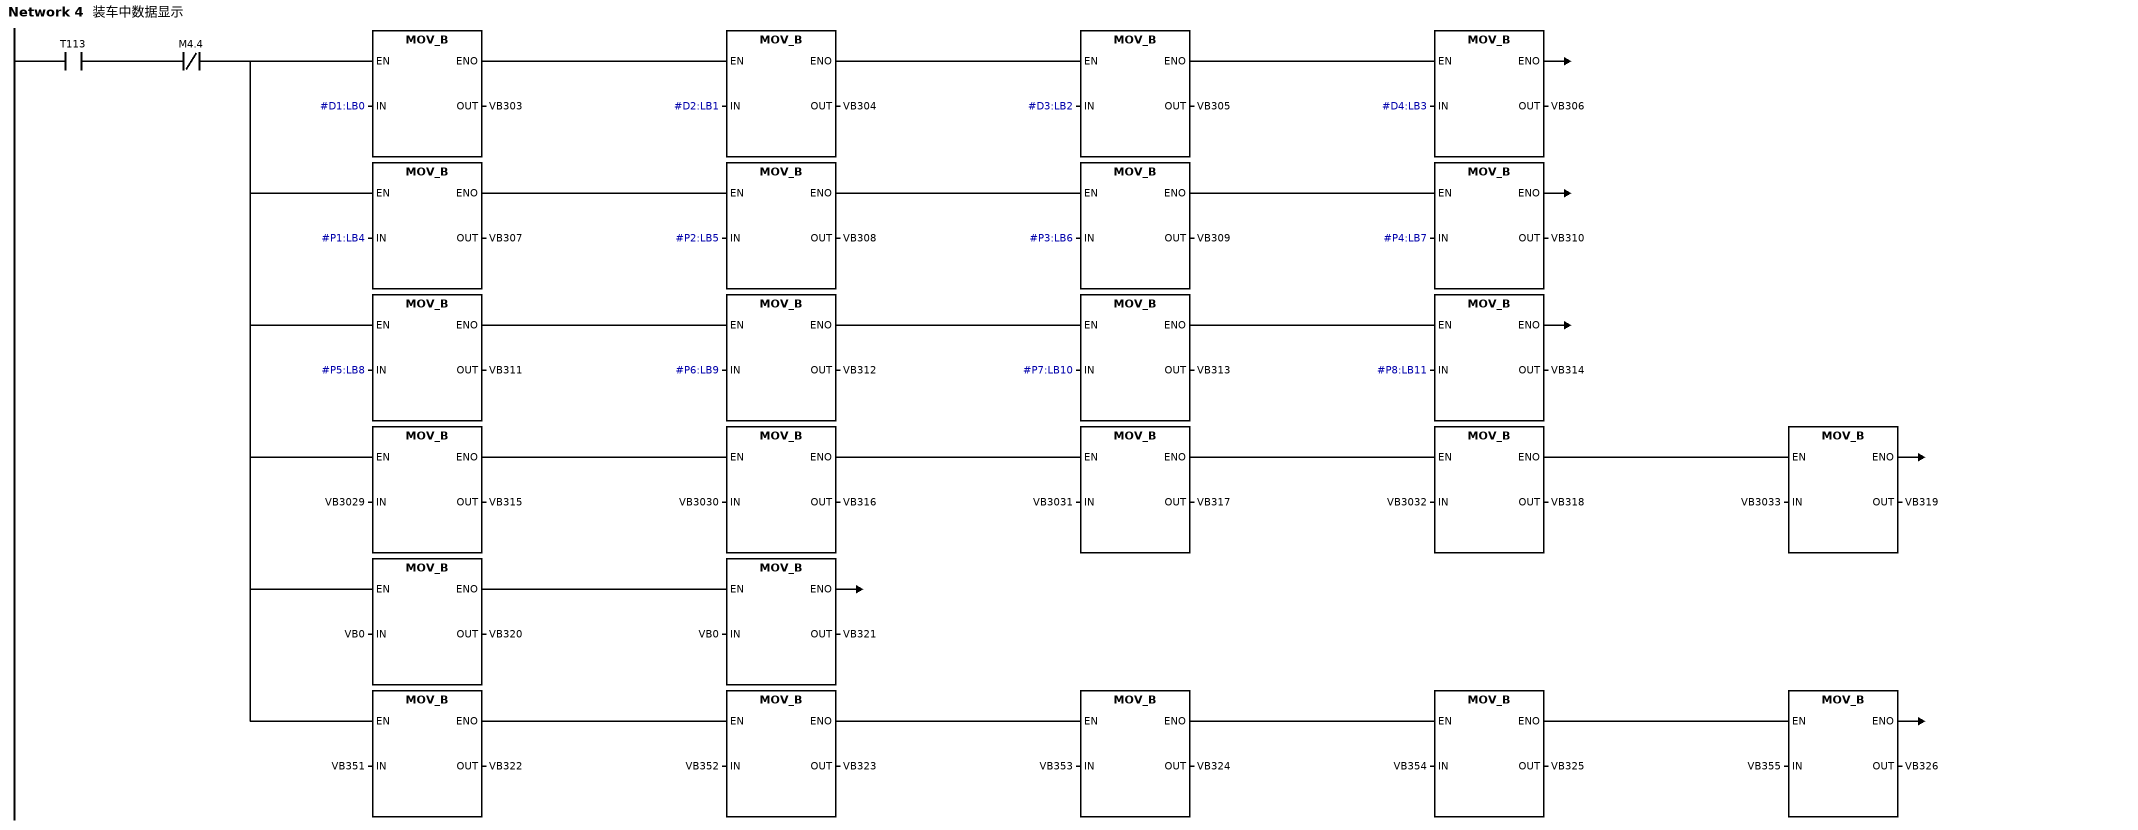
[picture p24: SBR13 networks 4-4]
Network 4 // 装车中数据显示
LD     T113
AN     M4.4
LPS
MOVB   #D1:LB0, VB303
AENO
MOVB   #D2:LB1, VB304
AENO
MOVB   #D3:LB2, VB305
AENO
MOVB   #D4:LB3, VB306
LRD
MOVB   #P1:LB4, VB307
AENO
MOVB   #P2:LB5, VB308
AENO
MOVB   #P3:LB6, VB309
AENO
MOVB   #P4:LB7, VB310
LRD
MOVB   #P5:LB8, VB311
AENO
MOVB   #P6:LB9, VB312
AENO
MOVB   #P7:LB10, VB313
AENO
MOVB   #P8:LB11, VB314
LRD
MOVB   VB3029, VB315
AENO
MOVB   VB3030, VB316
AENO
MOVB   VB3031, VB317
AENO
MOVB   VB3032, VB318
AENO
MOVB   VB3033, VB319
LRD
MOVB   VB0, VB320
AENO
MOVB   VB0, VB321
LPP
MOVB   VB351, VB322
AENO
MOVB   VB352, VB323
AENO
MOVB   VB353, VB324
AENO
MOVB   VB354, VB325
AENO
MOVB   VB355, VB326
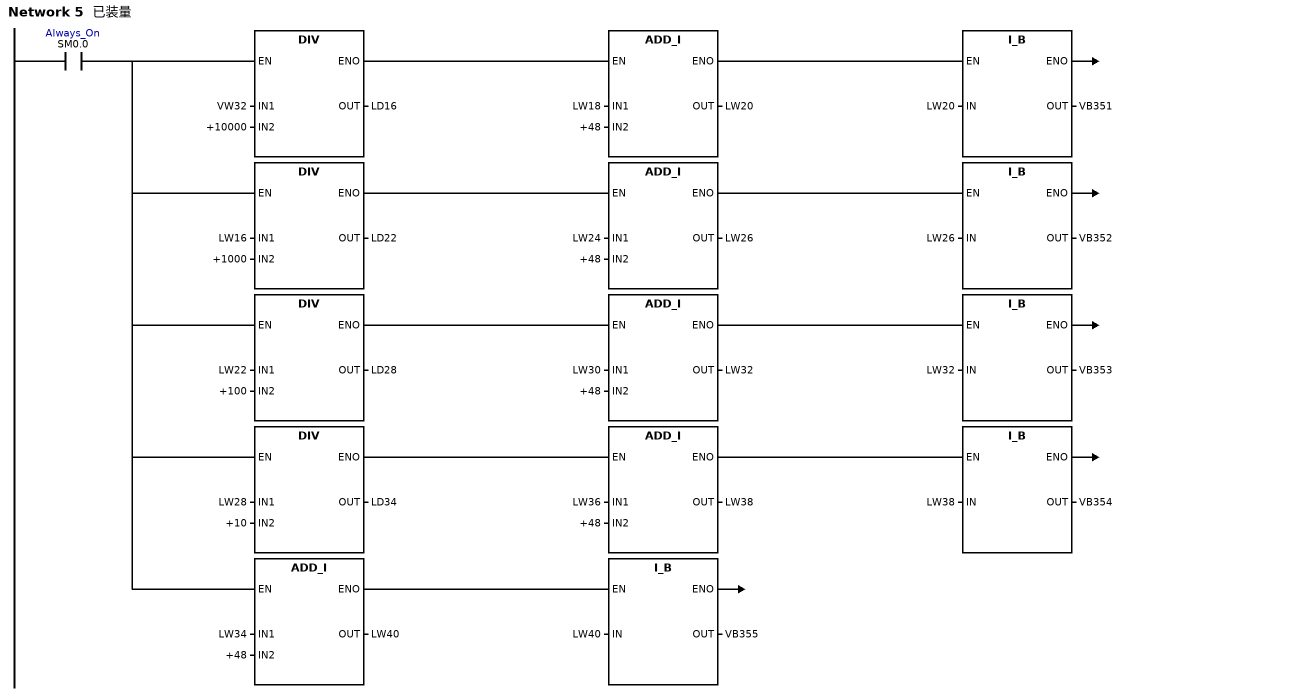
Network 5 // 已装量
LD     Always_On:SM0.0
LPS
MOVW   VW32, LW18
AENO
DIV    +10000, LD16
AENO
MOVW   LW18, LW20
AENO
+I     +48, LW20
AENO
ITB    LW20, VB351
LRD
MOVW   LW16, LW24
AENO
DIV    +1000, LD22
AENO
MOVW   LW24, LW26
AENO
+I     +48, LW26
AENO
ITB    LW26, VB352
LRD
MOVW   LW22, LW30
AENO
DIV    +100, LD28
AENO
MOVW   LW30, LW32
AENO
+I     +48, LW32
AENO
ITB    LW32, VB353
LRD
MOVW   LW28, LW36
AENO
DIV    +10, LD34
AENO
MOVW   LW36, LW38
AENO
+I     +48, LW38
AENO
ITB    LW38, VB354
LPP
MOVW   LW34, LW40
AENO
+I     +48, LW40
AENO
ITB    LW40, VB355
END_SUBROUTINE_BLOCK

SUBROUTINE_BLOCK LED4:SBR14
TITLE=
VAR_INPUT
D1:BYTE;	// LB0 
D2:BYTE;	// LB1 
D3:BYTE;	// LB2 
D4:BYTE;	// LB3 
P1:BYTE;	// LB4 
P2:BYTE;	// LB5 
P3:BYTE;	// LB6 
P4:BYTE;	// LB7 
P5:BYTE;	// LB8 
P6:BYTE;	// LB9 
P7:BYTE;	// LB10 
P8:BYTE;	// LB11 
RUN:WORD;	// LW12 
END_VAR
BEGIN
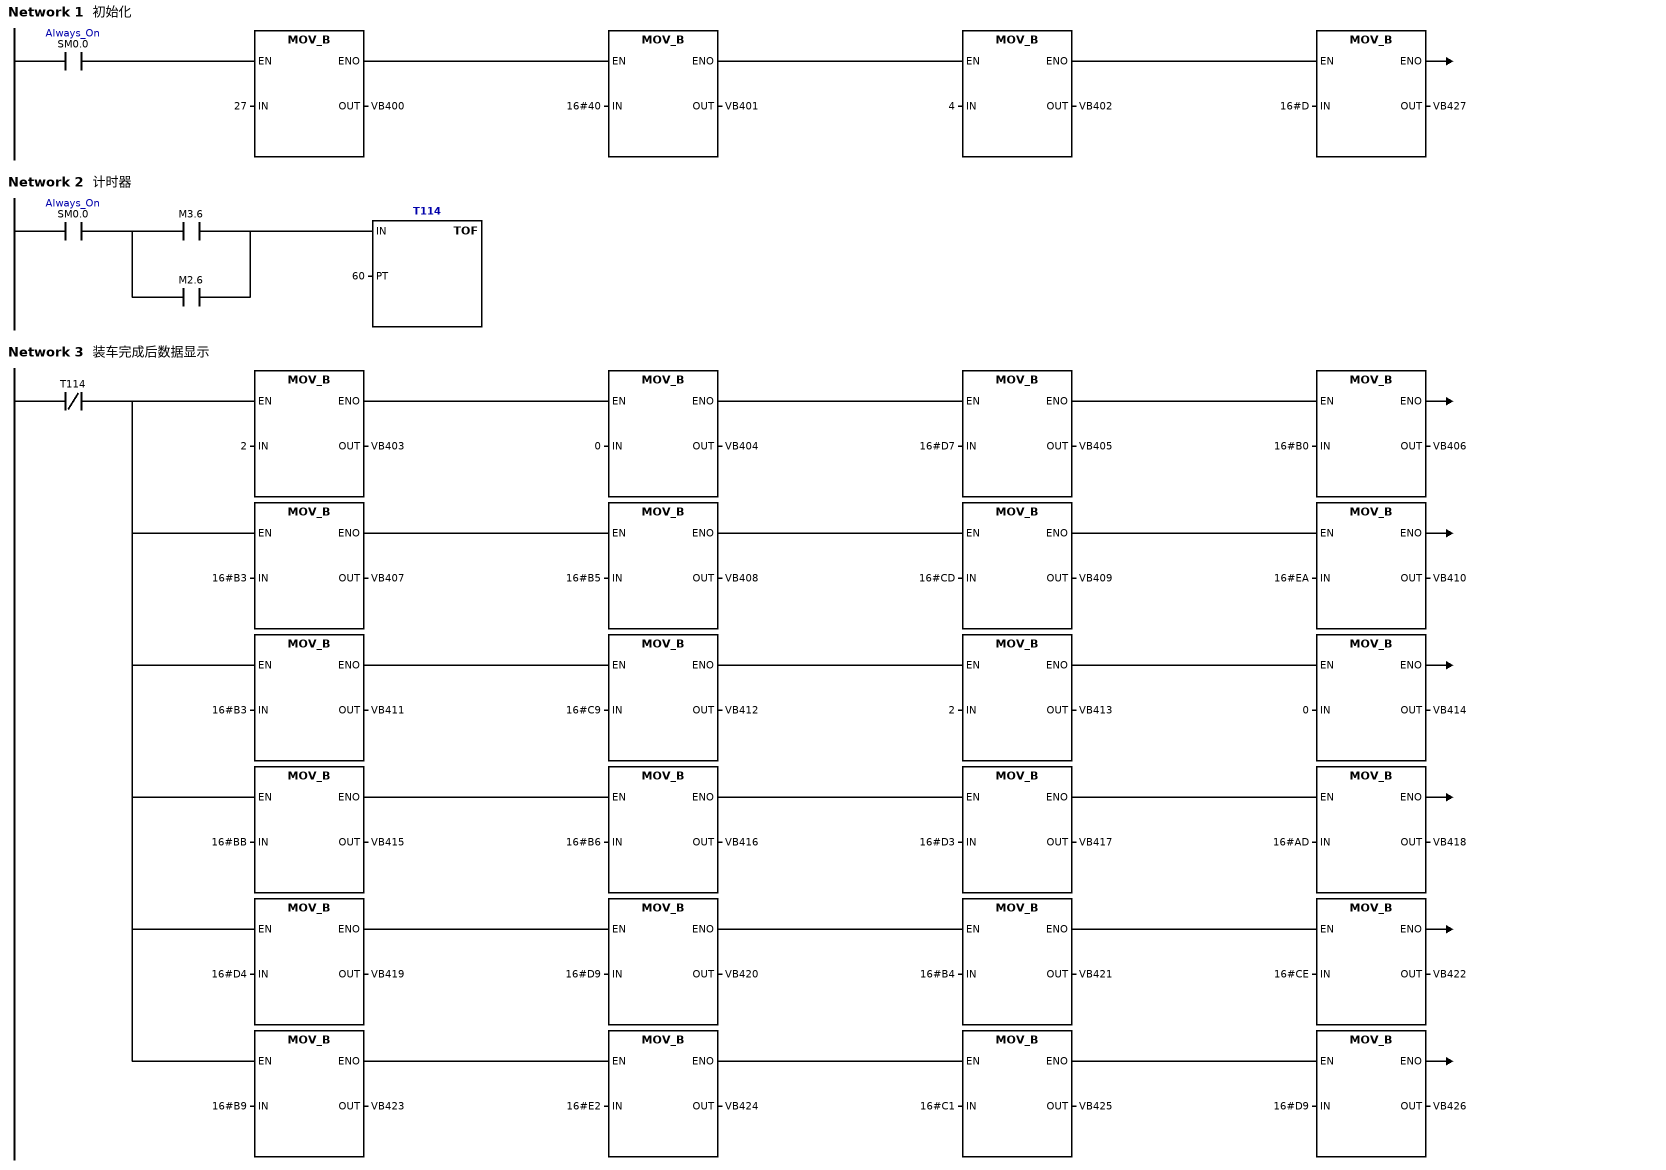
Network 1 // 初始化
LD     Always_On:SM0.0
MOVB   27, VB400
AENO
MOVB   16#40, VB401
AENO
MOVB   4, VB402
AENO
MOVB   16#D, VB427
Network 2 // 计时器
LD     Always_On:SM0.0
LD     M3.6
O      M2.6
ALD
TOF    T114, 60
Network 3 // 装车完成后数据显示
LDN    T114
LPS
MOVB   2, VB403
AENO
MOVB   0, VB404
AENO
MOVB   16#D7, VB405
AENO
MOVB   16#B0, VB406
LRD
MOVB   16#B3, VB407
AENO
MOVB   16#B5, VB408
AENO
MOVB   16#CD, VB409
AENO
MOVB   16#EA, VB410
LRD
MOVB   16#B3, VB411
AENO
MOVB   16#C9, VB412
AENO
MOVB   2, VB413
AENO
MOVB   0, VB414
LRD
MOVB   16#BB, VB415
AENO
MOVB   16#B6, VB416
AENO
MOVB   16#D3, VB417
AENO
MOVB   16#AD, VB418
LRD
MOVB   16#D4, VB419
AENO
MOVB   16#D9, VB420
AENO
MOVB   16#B4, VB421
AENO
MOVB   16#CE, VB422
LPP
MOVB   16#B9, VB423
AENO
MOVB   16#E2, VB424
AENO
MOVB   16#C1, VB425
AENO
MOVB   16#D9, VB426
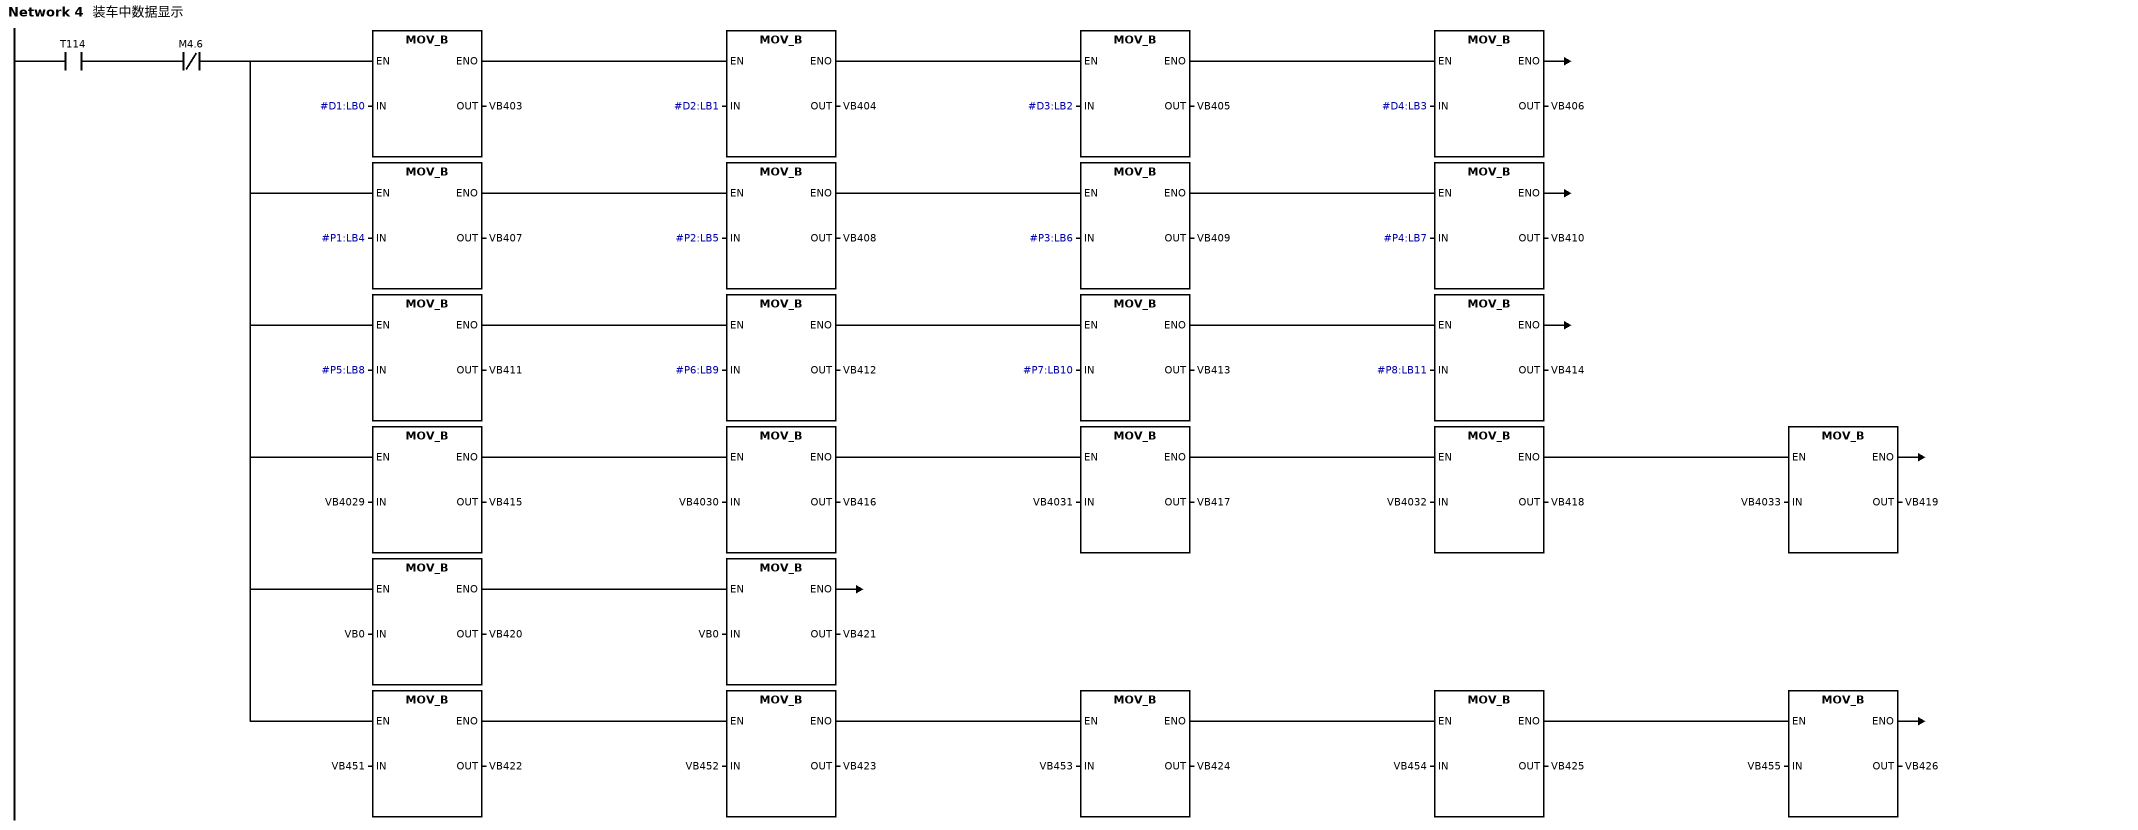
Network 4 // 装车中数据显示
LD     T114
AN     M4.6
LPS
MOVB   #D1:LB0, VB403
AENO
MOVB   #D2:LB1, VB404
AENO
MOVB   #D3:LB2, VB405
AENO
MOVB   #D4:LB3, VB406
LRD
MOVB   #P1:LB4, VB407
AENO
MOVB   #P2:LB5, VB408
AENO
MOVB   #P3:LB6, VB409
AENO
MOVB   #P4:LB7, VB410
LRD
MOVB   #P5:LB8, VB411
AENO
MOVB   #P6:LB9, VB412
AENO
MOVB   #P7:LB10, VB413
AENO
MOVB   #P8:LB11, VB414
LRD
MOVB   VB4029, VB415
AENO
MOVB   VB4030, VB416
AENO
MOVB   VB4031, VB417
AENO
MOVB   VB4032, VB418
AENO
MOVB   VB4033, VB419
LRD
MOVB   VB0, VB420
AENO
MOVB   VB0, VB421
LPP
MOVB   VB451, VB422
AENO
MOVB   VB452, VB423
AENO
MOVB   VB453, VB424
AENO
MOVB   VB454, VB425
AENO
MOVB   VB455, VB426
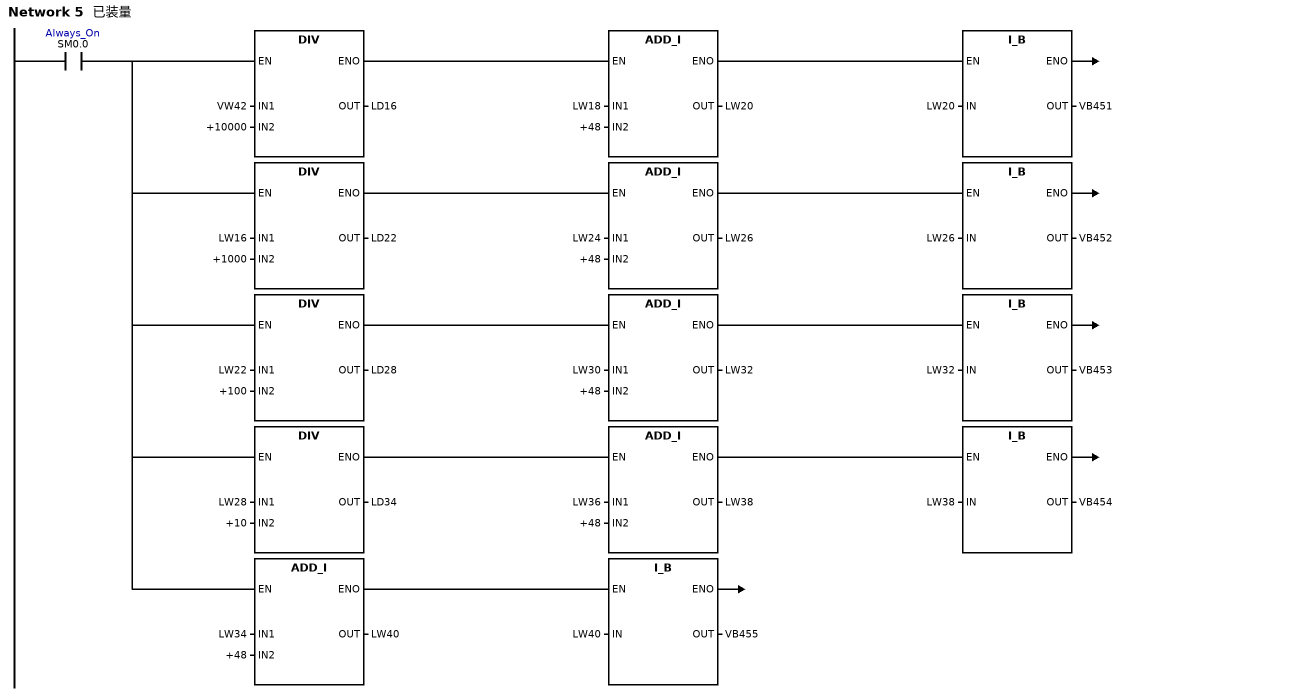
Network 5 // 已装量
LD     Always_On:SM0.0
LPS
MOVW   VW42, LW18
AENO
DIV    +10000, LD16
AENO
MOVW   LW18, LW20
AENO
+I     +48, LW20
AENO
ITB    LW20, VB451
LRD
MOVW   LW16, LW24
AENO
DIV    +1000, LD22
AENO
MOVW   LW24, LW26
AENO
+I     +48, LW26
AENO
ITB    LW26, VB452
LRD
MOVW   LW22, LW30
AENO
DIV    +100, LD28
AENO
MOVW   LW30, LW32
AENO
+I     +48, LW32
AENO
ITB    LW32, VB453
LRD
MOVW   LW28, LW36
AENO
DIV    +10, LD34
AENO
MOVW   LW36, LW38
AENO
+I     +48, LW38
AENO
ITB    LW38, VB454
LPP
MOVW   LW34, LW40
AENO
+I     +48, LW40
AENO
ITB    LW40, VB455
END_SUBROUTINE_BLOCK

SUBROUTINE_BLOCK N1收:SBR21
TITLE=
VAR_OUTPUT
总袋数1:WORD;	// LW0 
袋长1:WORD;	// LW2 
END_VAR
VAR
TEMP1:WORD;	// LW4 
TEMP2:WORD;	// LW6 
TEMP3:WORD;	// LW8 
TEMP4:WORD;	// LW10 
TEMP5:WORD;	// LW12 
TEMP6:WORD;	// LW14 
TEMP7:WORD;	// LW16 
TEMP8:WORD;	// LW18 
TEMP9:WORD;	// LW20 
TEMP10:WORD;	// LW22 
TEMP11:WORD;	// LW24 
TEMP12:WORD;	// LW26 
TEMP13:WORD;	// LW28 
TEMP14:WORD;	// LW30 
TEMP15:WORD;	// LW32 
TEMP16:WORD;	// LW34 
TEMP17:WORD;	// LW36 
TEMP18:WORD;	// LW38 
TEMP19:WORD;	// LW40 
TEMP20:WORD;	// LW42 
TEMP21:WORD;	// LW44 
END_VAR
BEGIN
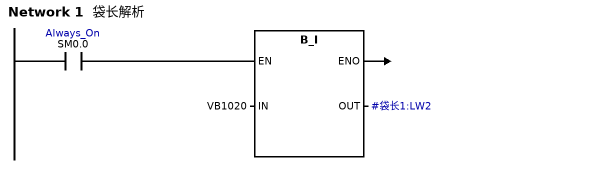
Network 1 // 袋长解析
LD     Always_On:SM0.0
BTI    VB1020, #袋长1:LW2
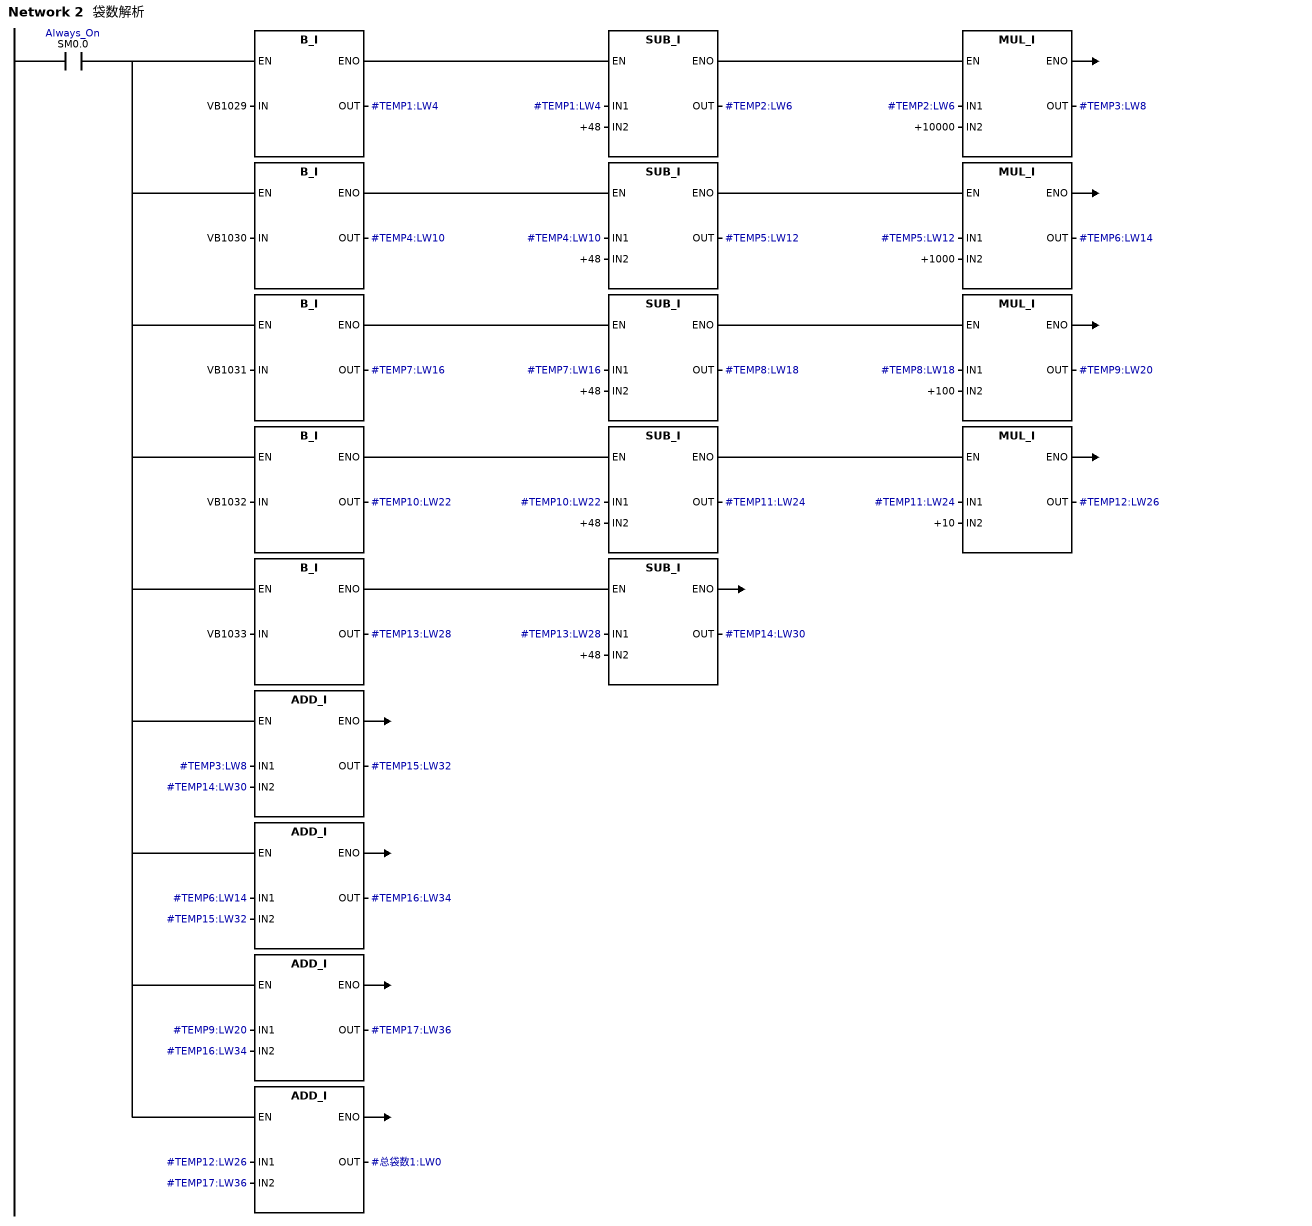
Network 2 // 袋数解析
LD     Always_On:SM0.0
LPS
BTI    VB1029, #TEMP1:LW4
AENO
MOVW   #TEMP1:LW4, #TEMP2:LW6
AENO
-I     +48, #TEMP2:LW6
AENO
MOVW   #TEMP2:LW6, #TEMP3:LW8
*I     +10000, #TEMP3:LW8
LRD
BTI    VB1030, #TEMP4:LW10
AENO
MOVW   #TEMP4:LW10, #TEMP5:LW12
AENO
-I     +48, #TEMP5:LW12
AENO
MOVW   #TEMP5:LW12, #TEMP6:LW14
*I     +1000, #TEMP6:LW14
LRD
BTI    VB1031, #TEMP7:LW16
AENO
MOVW   #TEMP7:LW16, #TEMP8:LW18
AENO
-I     +48, #TEMP8:LW18
AENO
MOVW   #TEMP8:LW18, #TEMP9:LW20
*I     +100, #TEMP9:LW20
LRD
BTI    VB1032, #TEMP10:LW22
AENO
MOVW   #TEMP10:LW22, #TEMP11:LW24
AENO
-I     +48, #TEMP11:LW24
AENO
MOVW   #TEMP11:LW24, #TEMP12:LW26
*I     +10, #TEMP12:LW26
LRD
BTI    VB1033, #TEMP13:LW28
AENO
MOVW   #TEMP13:LW28, #TEMP14:LW30
-I     +48, #TEMP14:LW30
LRD
MOVW   #TEMP3:LW8, #TEMP15:LW32
+I     #TEMP14:LW30, #TEMP15:LW32
LRD
MOVW   #TEMP6:LW14, #TEMP16:LW34
+I     #TEMP15:LW32, #TEMP16:LW34
LRD
MOVW   #TEMP9:LW20, #TEMP17:LW36
+I     #TEMP16:LW34, #TEMP17:LW36
LPP
MOVW   #TEMP12:LW26, #总袋数1:LW0
+I     #TEMP17:LW36, #总袋数1:LW0
END_SUBROUTINE_BLOCK

SUBROUTINE_BLOCK N2收:SBR22
TITLE=
VAR_OUTPUT
总袋数1:WORD;	// LW0 
袋长1:WORD;	// LW2 
END_VAR
VAR
TEMP1:WORD;	// LW4 
TEMP2:WORD;	// LW6 
TEMP3:WORD;	// LW8 
TEMP4:WORD;	// LW10 
TEMP5:WORD;	// LW12 
TEMP6:WORD;	// LW14 
TEMP7:WORD;	// LW16 
TEMP8:WORD;	// LW18 
TEMP9:WORD;	// LW20 
TEMP10:WORD;	// LW22 
TEMP11:WORD;	// LW24 
TEMP12:WORD;	// LW26 
TEMP13:WORD;	// LW28 
TEMP14:WORD;	// LW30 
TEMP15:WORD;	// LW32 
TEMP16:WORD;	// LW34 
TEMP17:WORD;	// LW36 
TEMP18:WORD;	// LW38 
TEMP19:WORD;	// LW40 
TEMP20:WORD;	// LW42 
TEMP21:WORD;	// LW44 
END_VAR
BEGIN
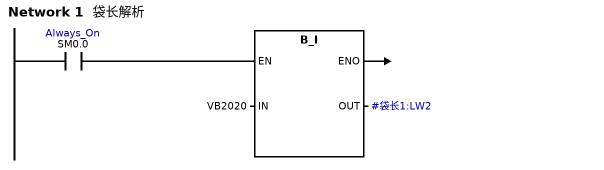
Network 1 // 袋长解析
LD     Always_On:SM0.0
BTI    VB2020, #袋长1:LW2
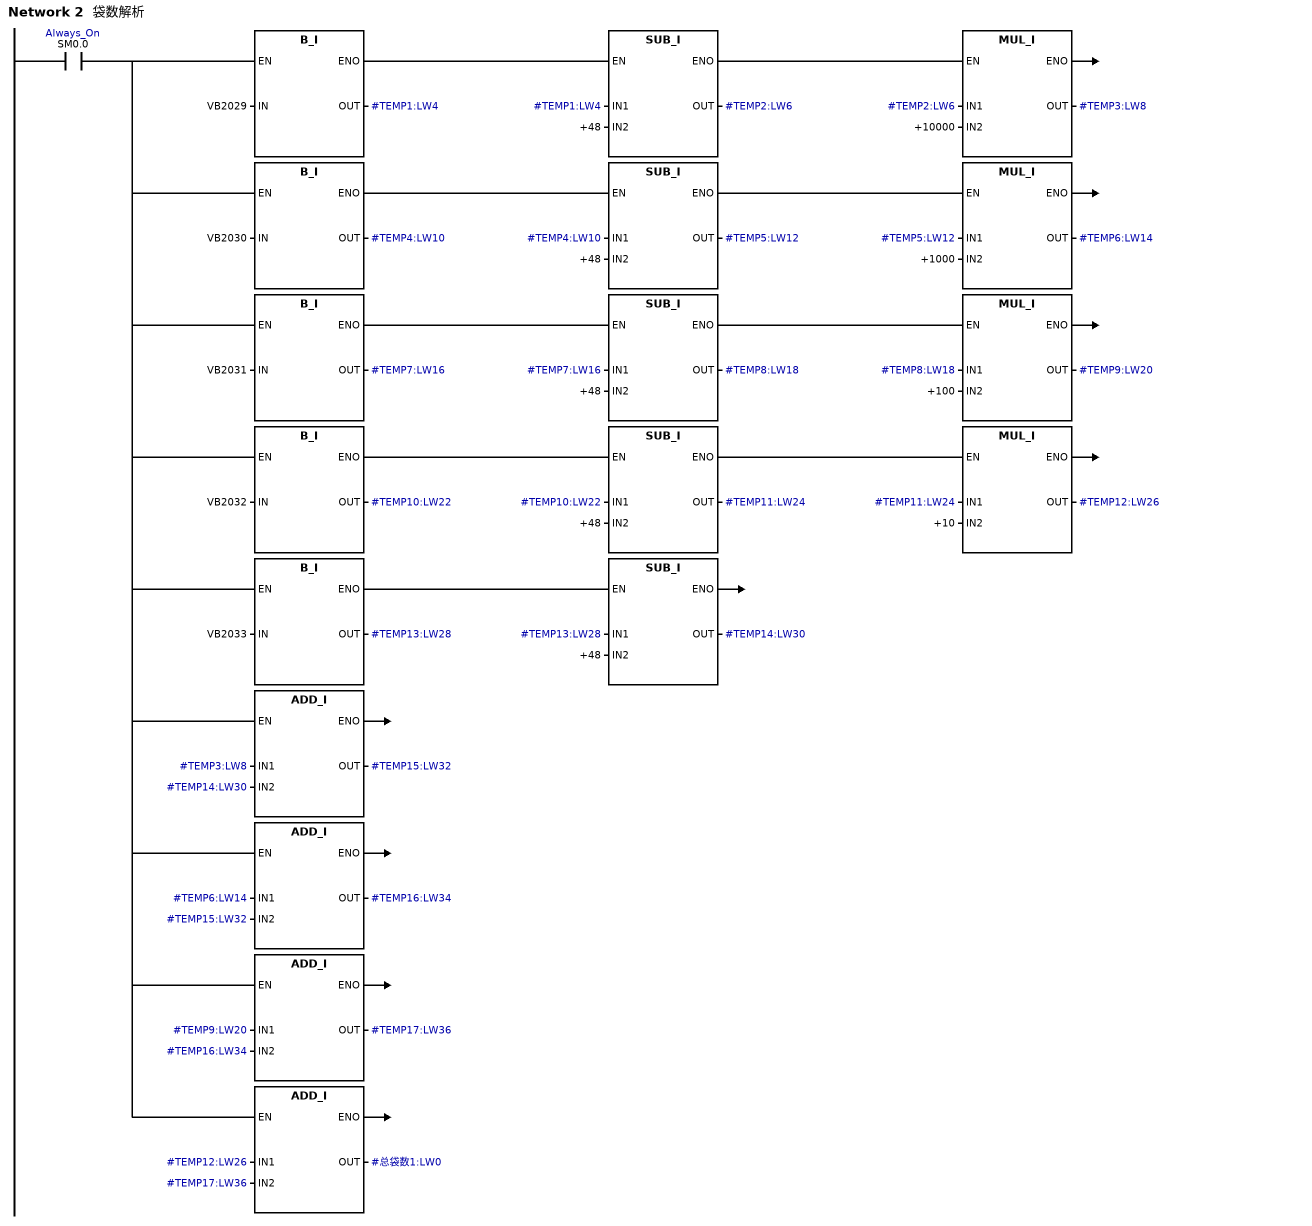
Network 2 // 袋数解析
LD     Always_On:SM0.0
LPS
BTI    VB2029, #TEMP1:LW4
AENO
MOVW   #TEMP1:LW4, #TEMP2:LW6
AENO
-I     +48, #TEMP2:LW6
AENO
MOVW   #TEMP2:LW6, #TEMP3:LW8
*I     +10000, #TEMP3:LW8
LRD
BTI    VB2030, #TEMP4:LW10
AENO
MOVW   #TEMP4:LW10, #TEMP5:LW12
AENO
-I     +48, #TEMP5:LW12
AENO
MOVW   #TEMP5:LW12, #TEMP6:LW14
*I     +1000, #TEMP6:LW14
LRD
BTI    VB2031, #TEMP7:LW16
AENO
MOVW   #TEMP7:LW16, #TEMP8:LW18
AENO
-I     +48, #TEMP8:LW18
AENO
MOVW   #TEMP8:LW18, #TEMP9:LW20
*I     +100, #TEMP9:LW20
LRD
BTI    VB2032, #TEMP10:LW22
AENO
MOVW   #TEMP10:LW22, #TEMP11:LW24
AENO
-I     +48, #TEMP11:LW24
AENO
MOVW   #TEMP11:LW24, #TEMP12:LW26
*I     +10, #TEMP12:LW26
LRD
BTI    VB2033, #TEMP13:LW28
AENO
MOVW   #TEMP13:LW28, #TEMP14:LW30
-I     +48, #TEMP14:LW30
LRD
MOVW   #TEMP3:LW8, #TEMP15:LW32
+I     #TEMP14:LW30, #TEMP15:LW32
LRD
MOVW   #TEMP6:LW14, #TEMP16:LW34
+I     #TEMP15:LW32, #TEMP16:LW34
LRD
MOVW   #TEMP9:LW20, #TEMP17:LW36
+I     #TEMP16:LW34, #TEMP17:LW36
LPP
MOVW   #TEMP12:LW26, #总袋数1:LW0
+I     #TEMP17:LW36, #总袋数1:LW0
END_SUBROUTINE_BLOCK

SUBROUTINE_BLOCK N3收:SBR23
TITLE=
VAR_OUTPUT
总袋数1:WORD;	// LW0 
袋长1:WORD;	// LW2 
END_VAR
VAR
TEMP1:WORD;	// LW4 
TEMP2:WORD;	// LW6 
TEMP3:WORD;	// LW8 
TEMP4:WORD;	// LW10 
TEMP5:WORD;	// LW12 
TEMP6:WORD;	// LW14 
TEMP7:WORD;	// LW16 
TEMP8:WORD;	// LW18 
TEMP9:WORD;	// LW20 
TEMP10:WORD;	// LW22 
TEMP11:WORD;	// LW24 
TEMP12:WORD;	// LW26 
TEMP13:WORD;	// LW28 
TEMP14:WORD;	// LW30 
TEMP15:WORD;	// LW32 
TEMP16:WORD;	// LW34 
TEMP17:WORD;	// LW36 
TEMP18:WORD;	// LW38 
TEMP19:WORD;	// LW40 
TEMP20:WORD;	// LW42 
TEMP21:WORD;	// LW44 
END_VAR
BEGIN
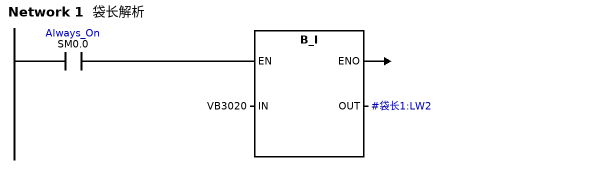
Network 1 // 袋长解析
LD     Always_On:SM0.0
BTI    VB3020, #袋长1:LW2
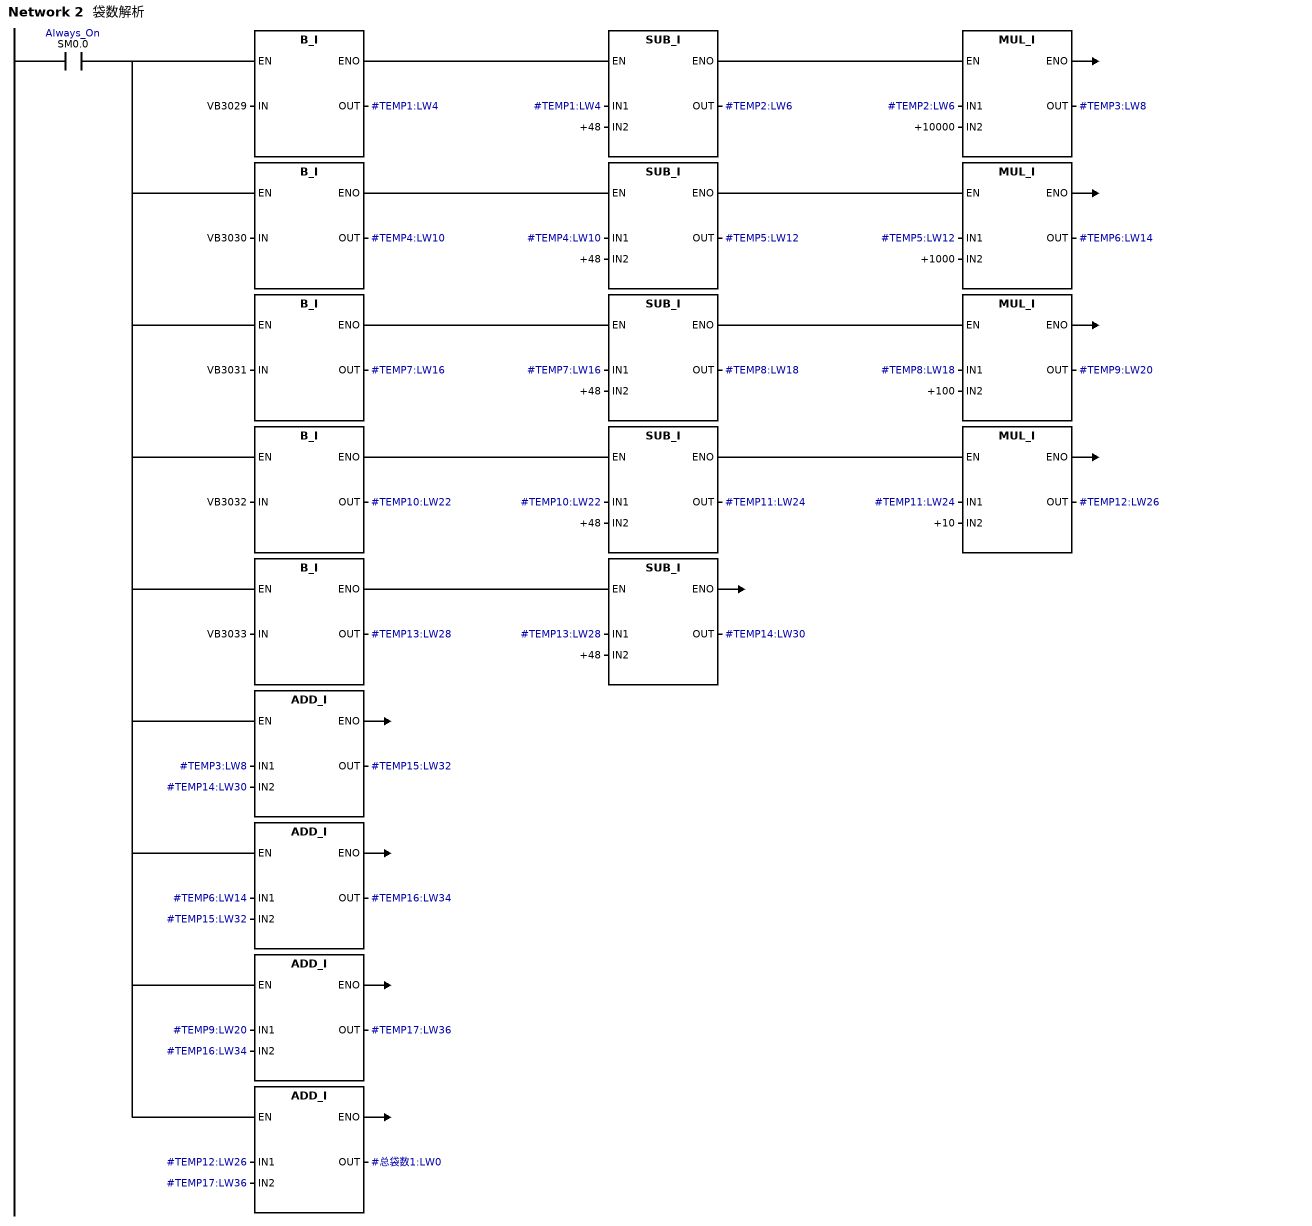
Network 2 // 袋数解析
LD     Always_On:SM0.0
LPS
BTI    VB3029, #TEMP1:LW4
AENO
MOVW   #TEMP1:LW4, #TEMP2:LW6
AENO
-I     +48, #TEMP2:LW6
AENO
MOVW   #TEMP2:LW6, #TEMP3:LW8
*I     +10000, #TEMP3:LW8
LRD
BTI    VB3030, #TEMP4:LW10
AENO
MOVW   #TEMP4:LW10, #TEMP5:LW12
AENO
-I     +48, #TEMP5:LW12
AENO
MOVW   #TEMP5:LW12, #TEMP6:LW14
*I     +1000, #TEMP6:LW14
LRD
BTI    VB3031, #TEMP7:LW16
AENO
MOVW   #TEMP7:LW16, #TEMP8:LW18
AENO
-I     +48, #TEMP8:LW18
AENO
MOVW   #TEMP8:LW18, #TEMP9:LW20
*I     +100, #TEMP9:LW20
LRD
BTI    VB3032, #TEMP10:LW22
AENO
MOVW   #TEMP10:LW22, #TEMP11:LW24
AENO
-I     +48, #TEMP11:LW24
AENO
MOVW   #TEMP11:LW24, #TEMP12:LW26
*I     +10, #TEMP12:LW26
LRD
BTI    VB3033, #TEMP13:LW28
AENO
MOVW   #TEMP13:LW28, #TEMP14:LW30
-I     +48, #TEMP14:LW30
LRD
MOVW   #TEMP3:LW8, #TEMP15:LW32
+I     #TEMP14:LW30, #TEMP15:LW32
LRD
MOVW   #TEMP6:LW14, #TEMP16:LW34
+I     #TEMP15:LW32, #TEMP16:LW34
LRD
MOVW   #TEMP9:LW20, #TEMP17:LW36
+I     #TEMP16:LW34, #TEMP17:LW36
LPP
MOVW   #TEMP12:LW26, #总袋数1:LW0
+I     #TEMP17:LW36, #总袋数1:LW0
END_SUBROUTINE_BLOCK

SUBROUTINE_BLOCK N4收:SBR24
TITLE=
VAR_OUTPUT
总袋数1:WORD;	// LW0 
袋长1:WORD;	// LW2 
END_VAR
VAR
TEMP1:WORD;	// LW4 
TEMP2:WORD;	// LW6 
TEMP3:WORD;	// LW8 
TEMP4:WORD;	// LW10 
TEMP5:WORD;	// LW12 
TEMP6:WORD;	// LW14 
TEMP7:WORD;	// LW16 
TEMP8:WORD;	// LW18 
TEMP9:WORD;	// LW20 
TEMP10:WORD;	// LW22 
TEMP11:WORD;	// LW24 
TEMP12:WORD;	// LW26 
TEMP13:WORD;	// LW28 
TEMP14:WORD;	// LW30 
TEMP15:WORD;	// LW32 
TEMP16:WORD;	// LW34 
TEMP17:WORD;	// LW36 
TEMP18:WORD;	// LW38 
TEMP19:WORD;	// LW40 
TEMP20:WORD;	// LW42 
TEMP21:WORD;	// LW44 
END_VAR
BEGIN
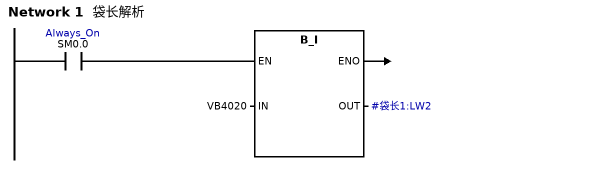
Network 1 // 袋长解析
LD     Always_On:SM0.0
BTI    VB4020, #袋长1:LW2
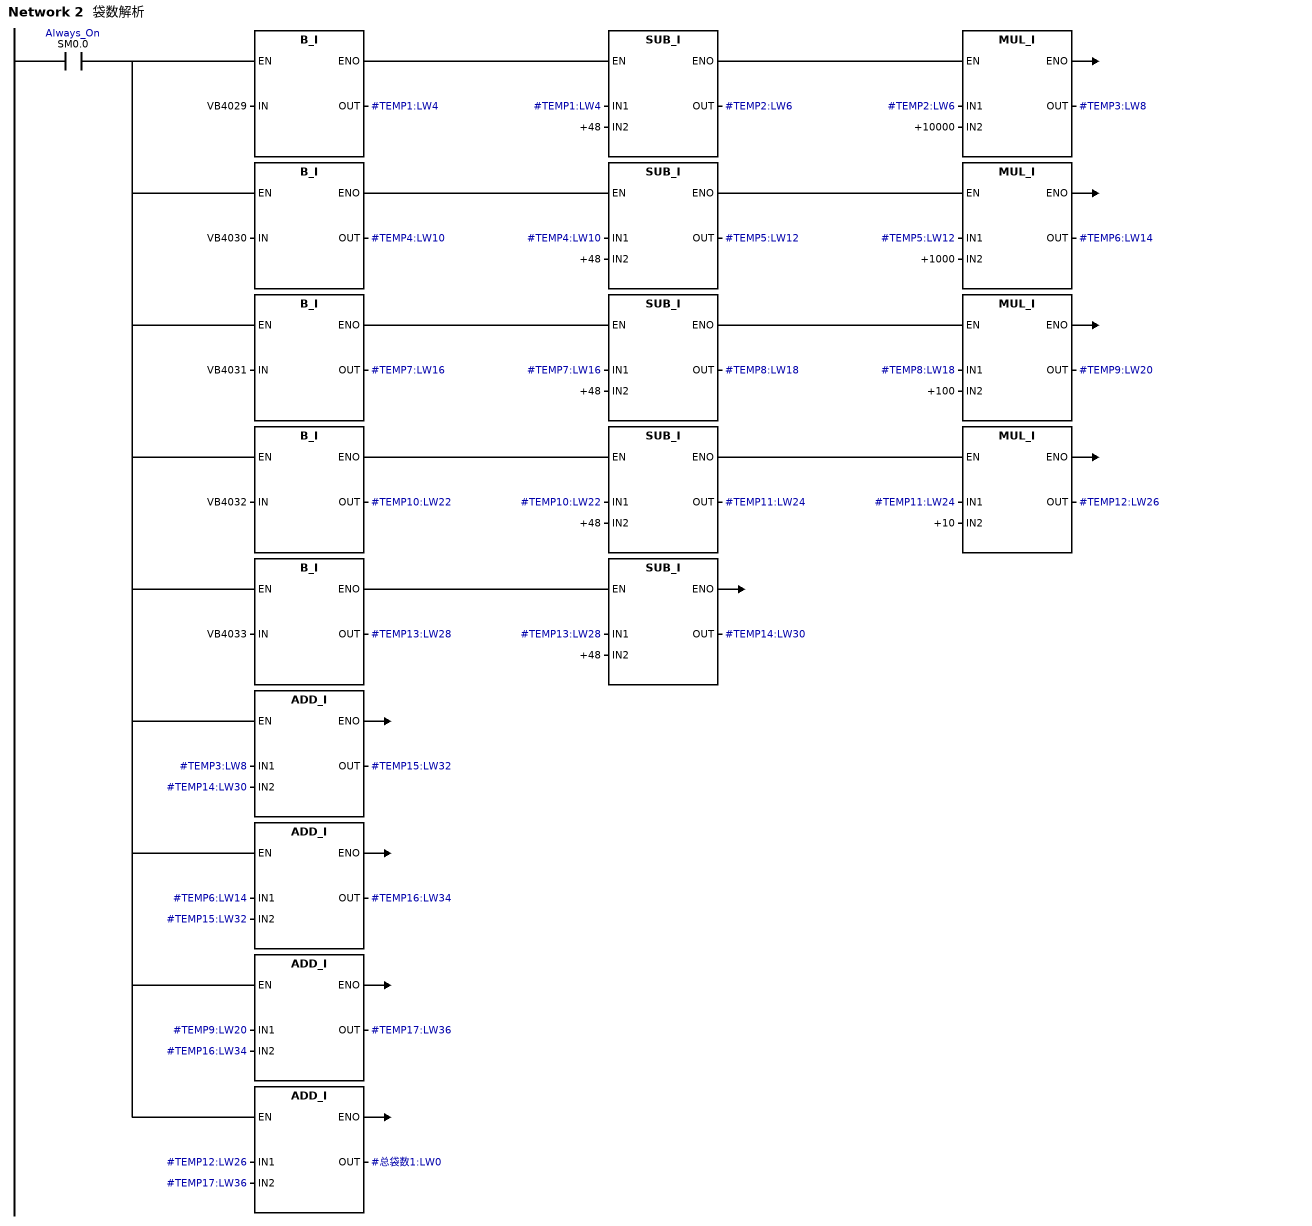
Network 2 // 袋数解析
LD     Always_On:SM0.0
LPS
BTI    VB4029, #TEMP1:LW4
AENO
MOVW   #TEMP1:LW4, #TEMP2:LW6
AENO
-I     +48, #TEMP2:LW6
AENO
MOVW   #TEMP2:LW6, #TEMP3:LW8
*I     +10000, #TEMP3:LW8
LRD
BTI    VB4030, #TEMP4:LW10
AENO
MOVW   #TEMP4:LW10, #TEMP5:LW12
AENO
-I     +48, #TEMP5:LW12
AENO
MOVW   #TEMP5:LW12, #TEMP6:LW14
*I     +1000, #TEMP6:LW14
LRD
BTI    VB4031, #TEMP7:LW16
AENO
MOVW   #TEMP7:LW16, #TEMP8:LW18
AENO
-I     +48, #TEMP8:LW18
AENO
MOVW   #TEMP8:LW18, #TEMP9:LW20
*I     +100, #TEMP9:LW20
LRD
BTI    VB4032, #TEMP10:LW22
AENO
MOVW   #TEMP10:LW22, #TEMP11:LW24
AENO
-I     +48, #TEMP11:LW24
AENO
MOVW   #TEMP11:LW24, #TEMP12:LW26
*I     +10, #TEMP12:LW26
LRD
BTI    VB4033, #TEMP13:LW28
AENO
MOVW   #TEMP13:LW28, #TEMP14:LW30
-I     +48, #TEMP14:LW30
LRD
MOVW   #TEMP3:LW8, #TEMP15:LW32
+I     #TEMP14:LW30, #TEMP15:LW32
LRD
MOVW   #TEMP6:LW14, #TEMP16:LW34
+I     #TEMP15:LW32, #TEMP16:LW34
LRD
MOVW   #TEMP9:LW20, #TEMP17:LW36
+I     #TEMP16:LW34, #TEMP17:LW36
LPP
MOVW   #TEMP12:LW26, #总袋数1:LW0
+I     #TEMP17:LW36, #总袋数1:LW0
END_SUBROUTINE_BLOCK

SUBROUTINE_BLOCK GGLED1_2:SBR31
TITLE=子程序注释
VAR_INPUT
屏3地址:BYTE;	// LB0 
END_VAR
BEGIN
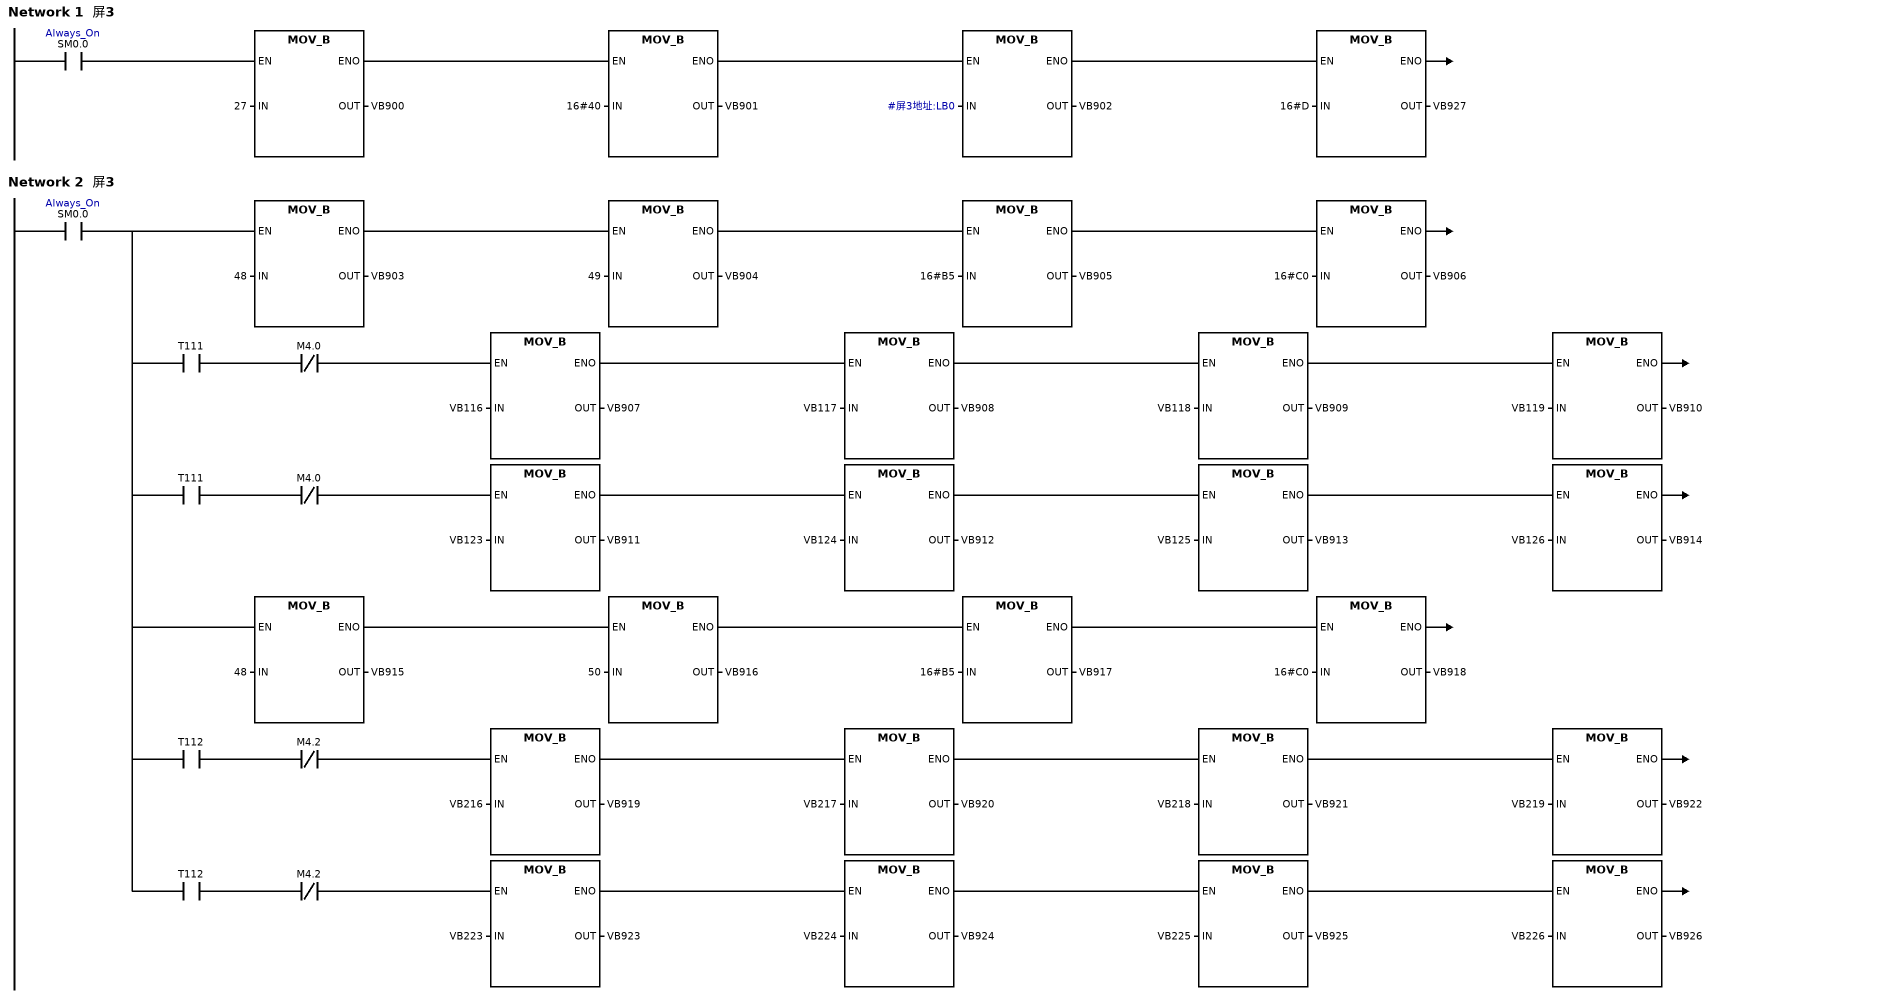
Network 1 // 屏3
LD     Always_On:SM0.0
MOVB   27, VB900
AENO
MOVB   16#40, VB901
AENO
MOVB   #屏3地址:LB0, VB902
AENO
MOVB   16#D, VB927
Network 2 // 屏3
LD     Always_On:SM0.0
LPS
MOVB   48, VB903
AENO
MOVB   49, VB904
AENO
MOVB   16#B5, VB905
AENO
MOVB   16#C0, VB906
LRD
A      T111
AN     M4.0
MOVB   VB116, VB907
AENO
MOVB   VB117, VB908
AENO
MOVB   VB118, VB909
AENO
MOVB   VB119, VB910
LRD
A      T111
AN     M4.0
MOVB   VB123, VB911
AENO
MOVB   VB124, VB912
AENO
MOVB   VB125, VB913
AENO
MOVB   VB126, VB914
LRD
MOVB   48, VB915
AENO
MOVB   50, VB916
AENO
MOVB   16#B5, VB917
AENO
MOVB   16#C0, VB918
LRD
A      T112
AN     M4.2
MOVB   VB216, VB919
AENO
MOVB   VB217, VB920
AENO
MOVB   VB218, VB921
AENO
MOVB   VB219, VB922
LPP
A      T112
AN     M4.2
MOVB   VB223, VB923
AENO
MOVB   VB224, VB924
AENO
MOVB   VB225, VB925
AENO
MOVB   VB226, VB926
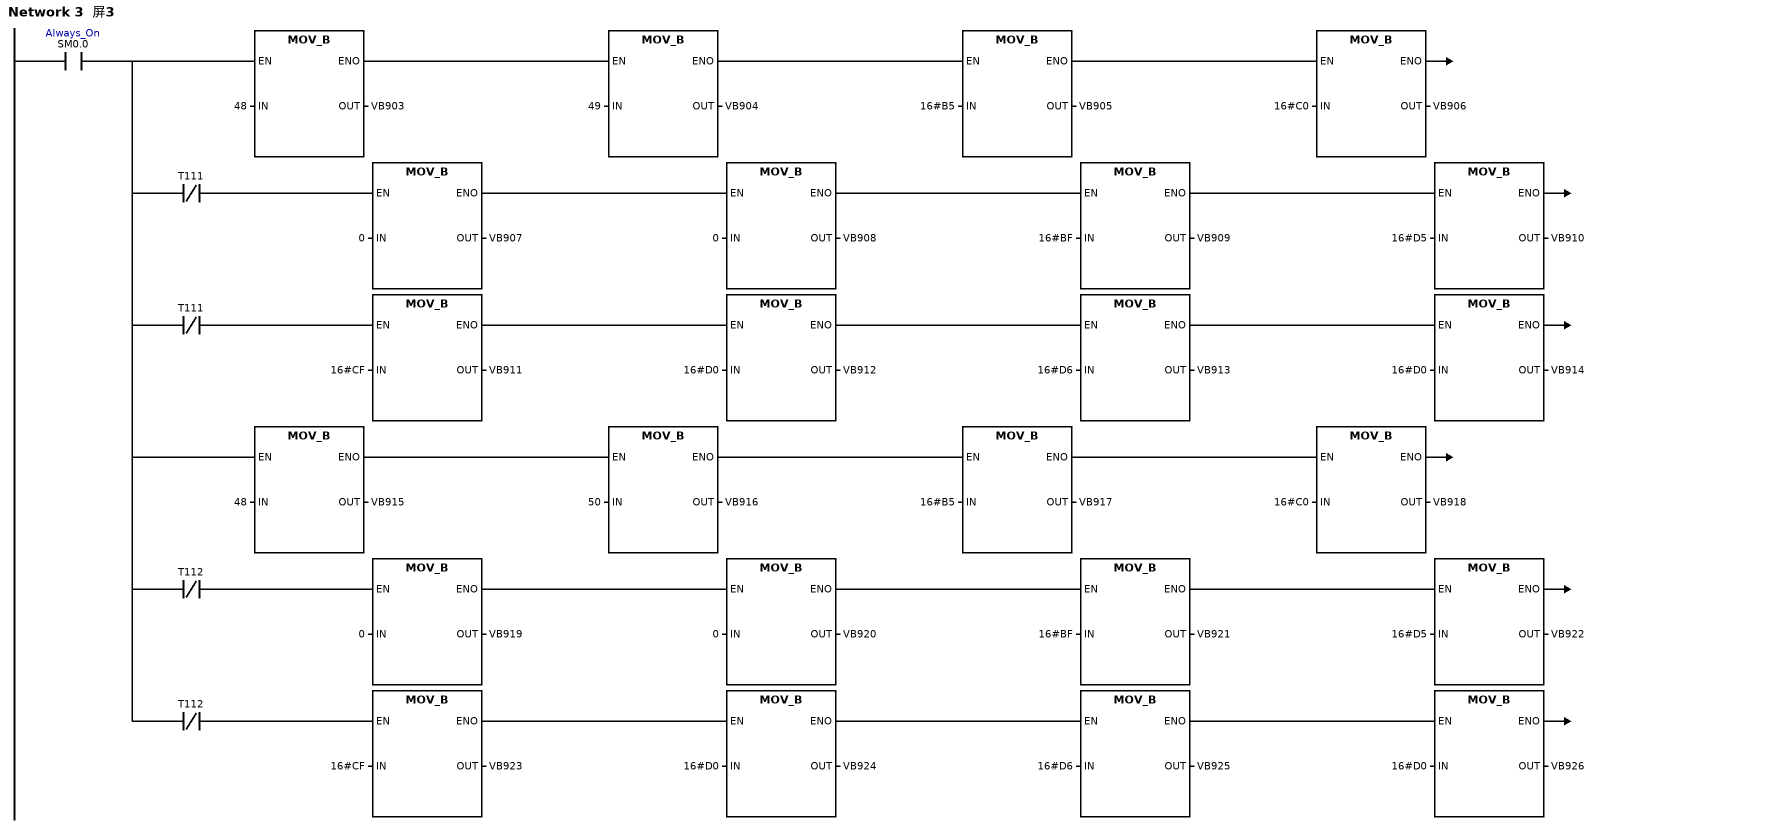
Network 3 // 屏3
LD     Always_On:SM0.0
LPS
MOVB   48, VB903
AENO
MOVB   49, VB904
AENO
MOVB   16#B5, VB905
AENO
MOVB   16#C0, VB906
LRD
AN     T111
MOVB   0, VB907
AENO
MOVB   0, VB908
AENO
MOVB   16#BF, VB909
AENO
MOVB   16#D5, VB910
LRD
AN     T111
MOVB   16#CF, VB911
AENO
MOVB   16#D0, VB912
AENO
MOVB   16#D6, VB913
AENO
MOVB   16#D0, VB914
LRD
MOVB   48, VB915
AENO
MOVB   50, VB916
AENO
MOVB   16#B5, VB917
AENO
MOVB   16#C0, VB918
LRD
AN     T112
MOVB   0, VB919
AENO
MOVB   0, VB920
AENO
MOVB   16#BF, VB921
AENO
MOVB   16#D5, VB922
LPP
AN     T112
MOVB   16#CF, VB923
AENO
MOVB   16#D0, VB924
AENO
MOVB   16#D6, VB925
AENO
MOVB   16#D0, VB926
END_SUBROUTINE_BLOCK

SUBROUTINE_BLOCK GGLED3_4:SBR32
TITLE=子程序注释
VAR_INPUT
屏3地址:BYTE;	// LB0 
END_VAR
BEGIN
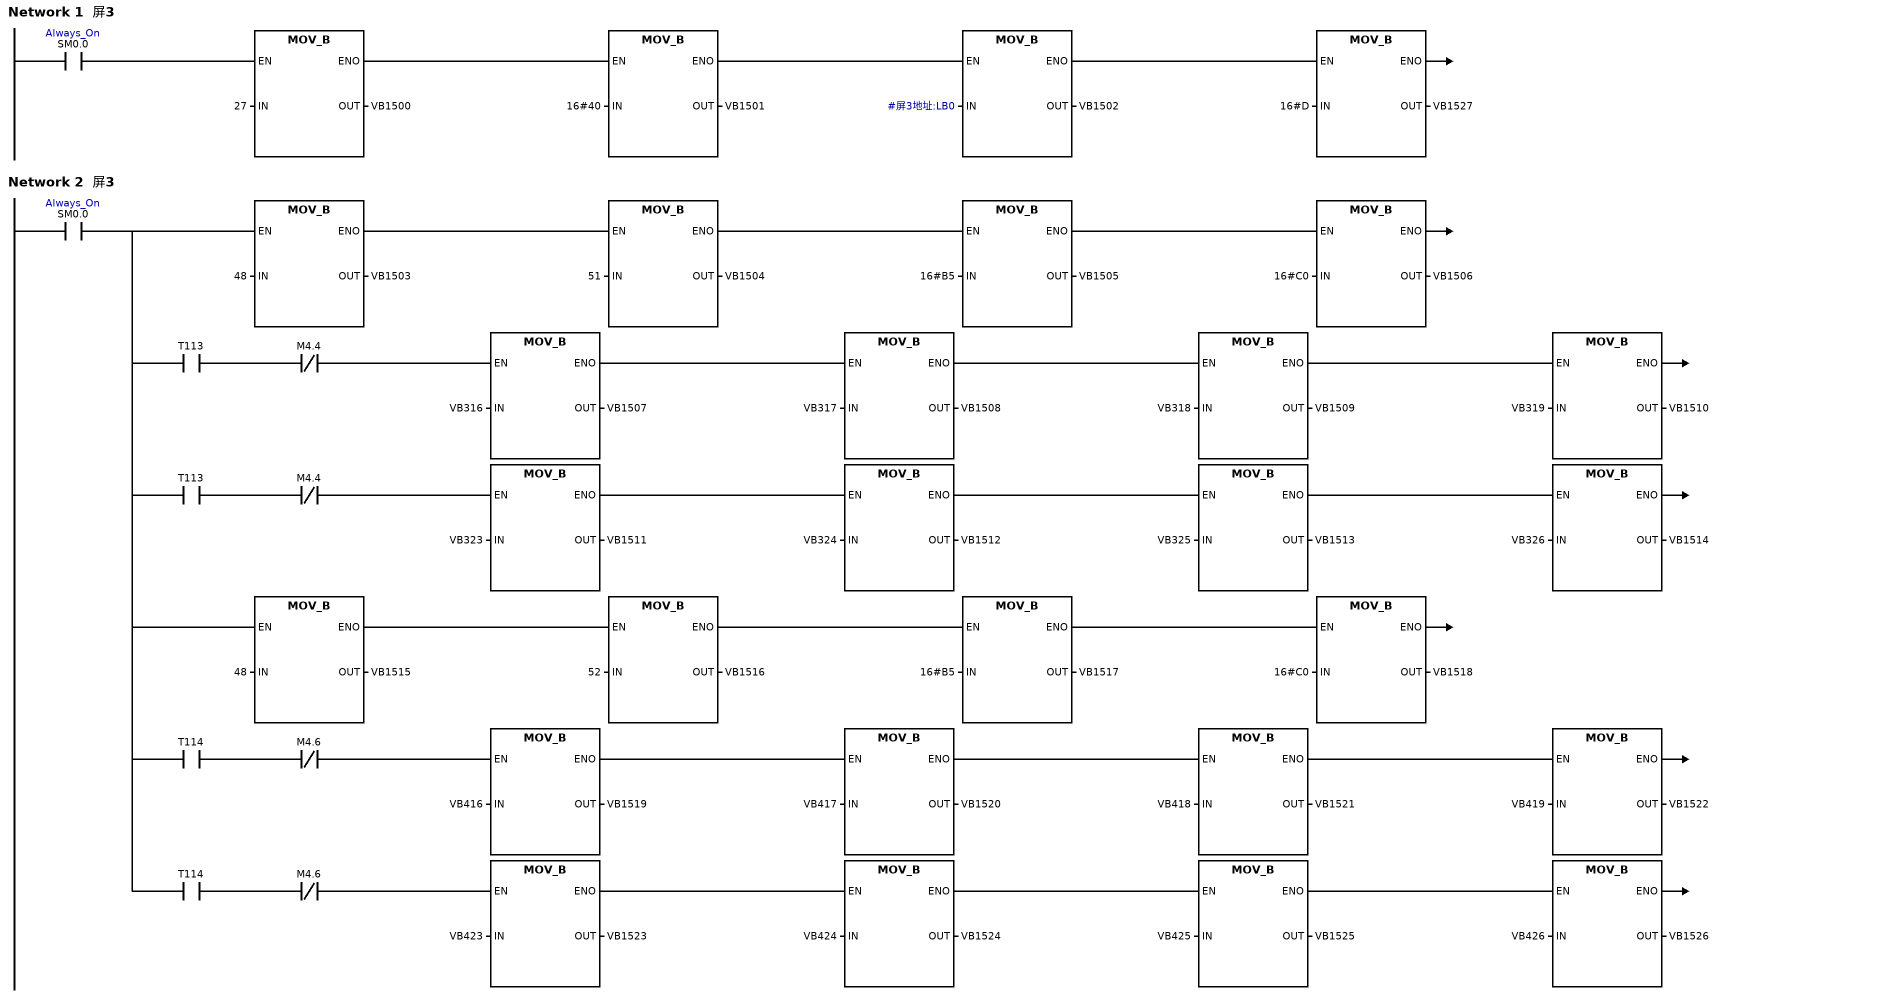
Network 1 // 屏3
LD     Always_On:SM0.0
MOVB   27, VB1500
AENO
MOVB   16#40, VB1501
AENO
MOVB   #屏3地址:LB0, VB1502
AENO
MOVB   16#D, VB1527
Network 2 // 屏3
LD     Always_On:SM0.0
LPS
MOVB   48, VB1503
AENO
MOVB   51, VB1504
AENO
MOVB   16#B5, VB1505
AENO
MOVB   16#C0, VB1506
LRD
A      T113
AN     M4.4
MOVB   VB316, VB1507
AENO
MOVB   VB317, VB1508
AENO
MOVB   VB318, VB1509
AENO
MOVB   VB319, VB1510
LRD
A      T113
AN     M4.4
MOVB   VB323, VB1511
AENO
MOVB   VB324, VB1512
AENO
MOVB   VB325, VB1513
AENO
MOVB   VB326, VB1514
LRD
MOVB   48, VB1515
AENO
MOVB   52, VB1516
AENO
MOVB   16#B5, VB1517
AENO
MOVB   16#C0, VB1518
LRD
A      T114
AN     M4.6
MOVB   VB416, VB1519
AENO
MOVB   VB417, VB1520
AENO
MOVB   VB418, VB1521
AENO
MOVB   VB419, VB1522
LPP
A      T114
AN     M4.6
MOVB   VB423, VB1523
AENO
MOVB   VB424, VB1524
AENO
MOVB   VB425, VB1525
AENO
MOVB   VB426, VB1526
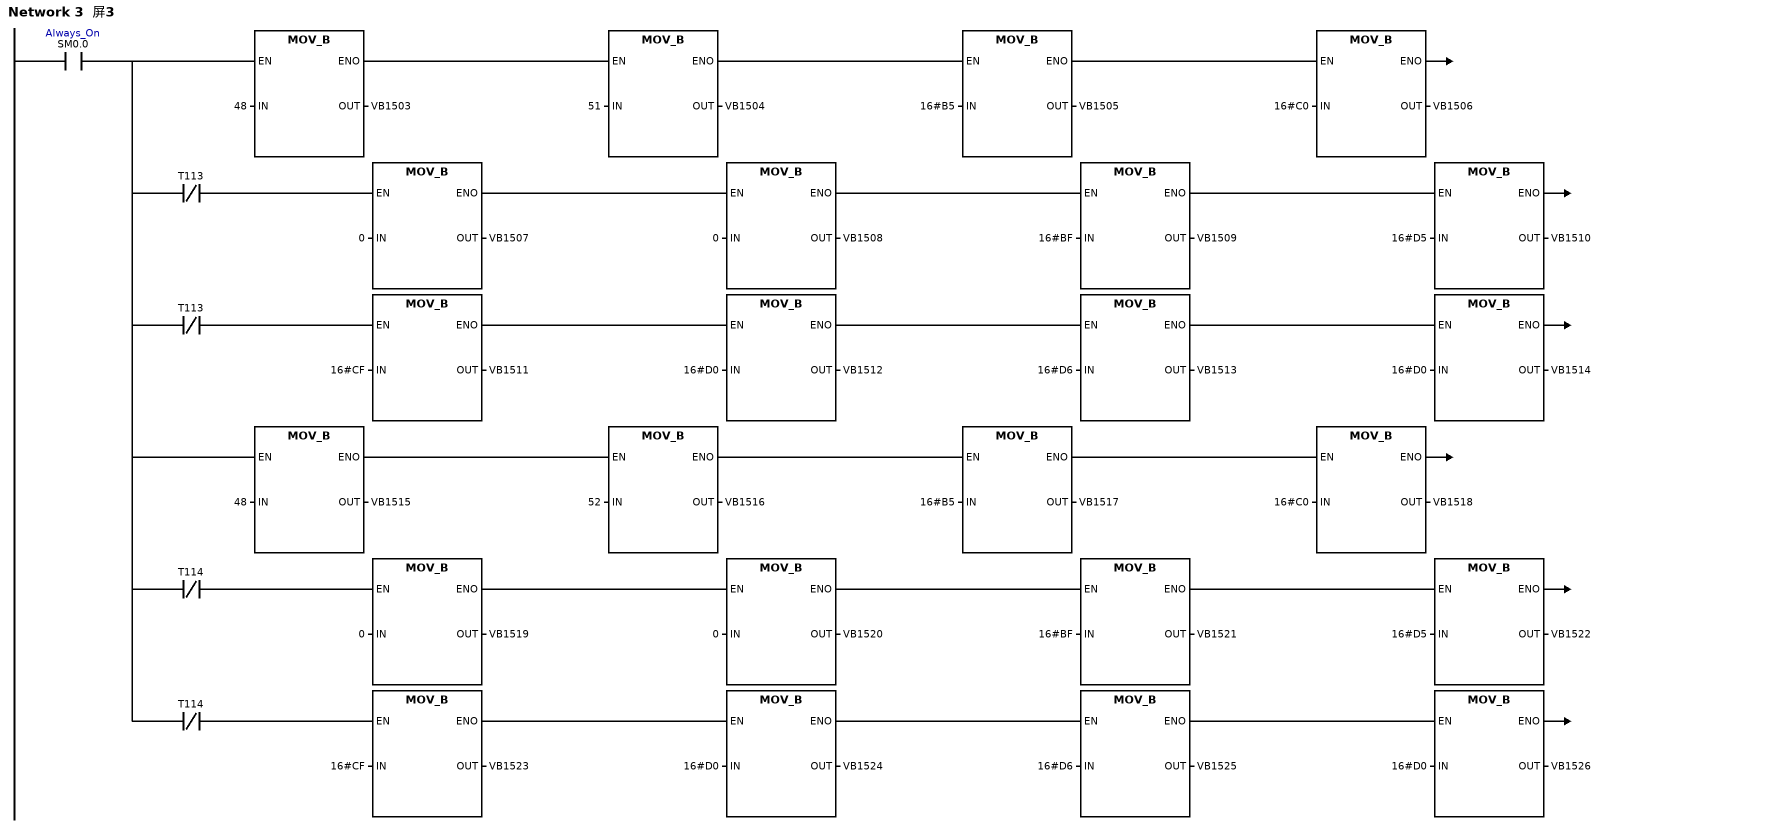
Network 3 // 屏3
LD     Always_On:SM0.0
LPS
MOVB   48, VB1503
AENO
MOVB   51, VB1504
AENO
MOVB   16#B5, VB1505
AENO
MOVB   16#C0, VB1506
LRD
AN     T113
MOVB   0, VB1507
AENO
MOVB   0, VB1508
AENO
MOVB   16#BF, VB1509
AENO
MOVB   16#D5, VB1510
LRD
AN     T113
MOVB   16#CF, VB1511
AENO
MOVB   16#D0, VB1512
AENO
MOVB   16#D6, VB1513
AENO
MOVB   16#D0, VB1514
LRD
MOVB   48, VB1515
AENO
MOVB   52, VB1516
AENO
MOVB   16#B5, VB1517
AENO
MOVB   16#C0, VB1518
LRD
AN     T114
MOVB   0, VB1519
AENO
MOVB   0, VB1520
AENO
MOVB   16#BF, VB1521
AENO
MOVB   16#D5, VB1522
LPP
AN     T114
MOVB   16#CF, VB1523
AENO
MOVB   16#D0, VB1524
AENO
MOVB   16#D6, VB1525
AENO
MOVB   16#D0, VB1526
END_SUBROUTINE_BLOCK

INTERRUPT_BLOCK RECEI:INT1
TITLE=
BEGIN
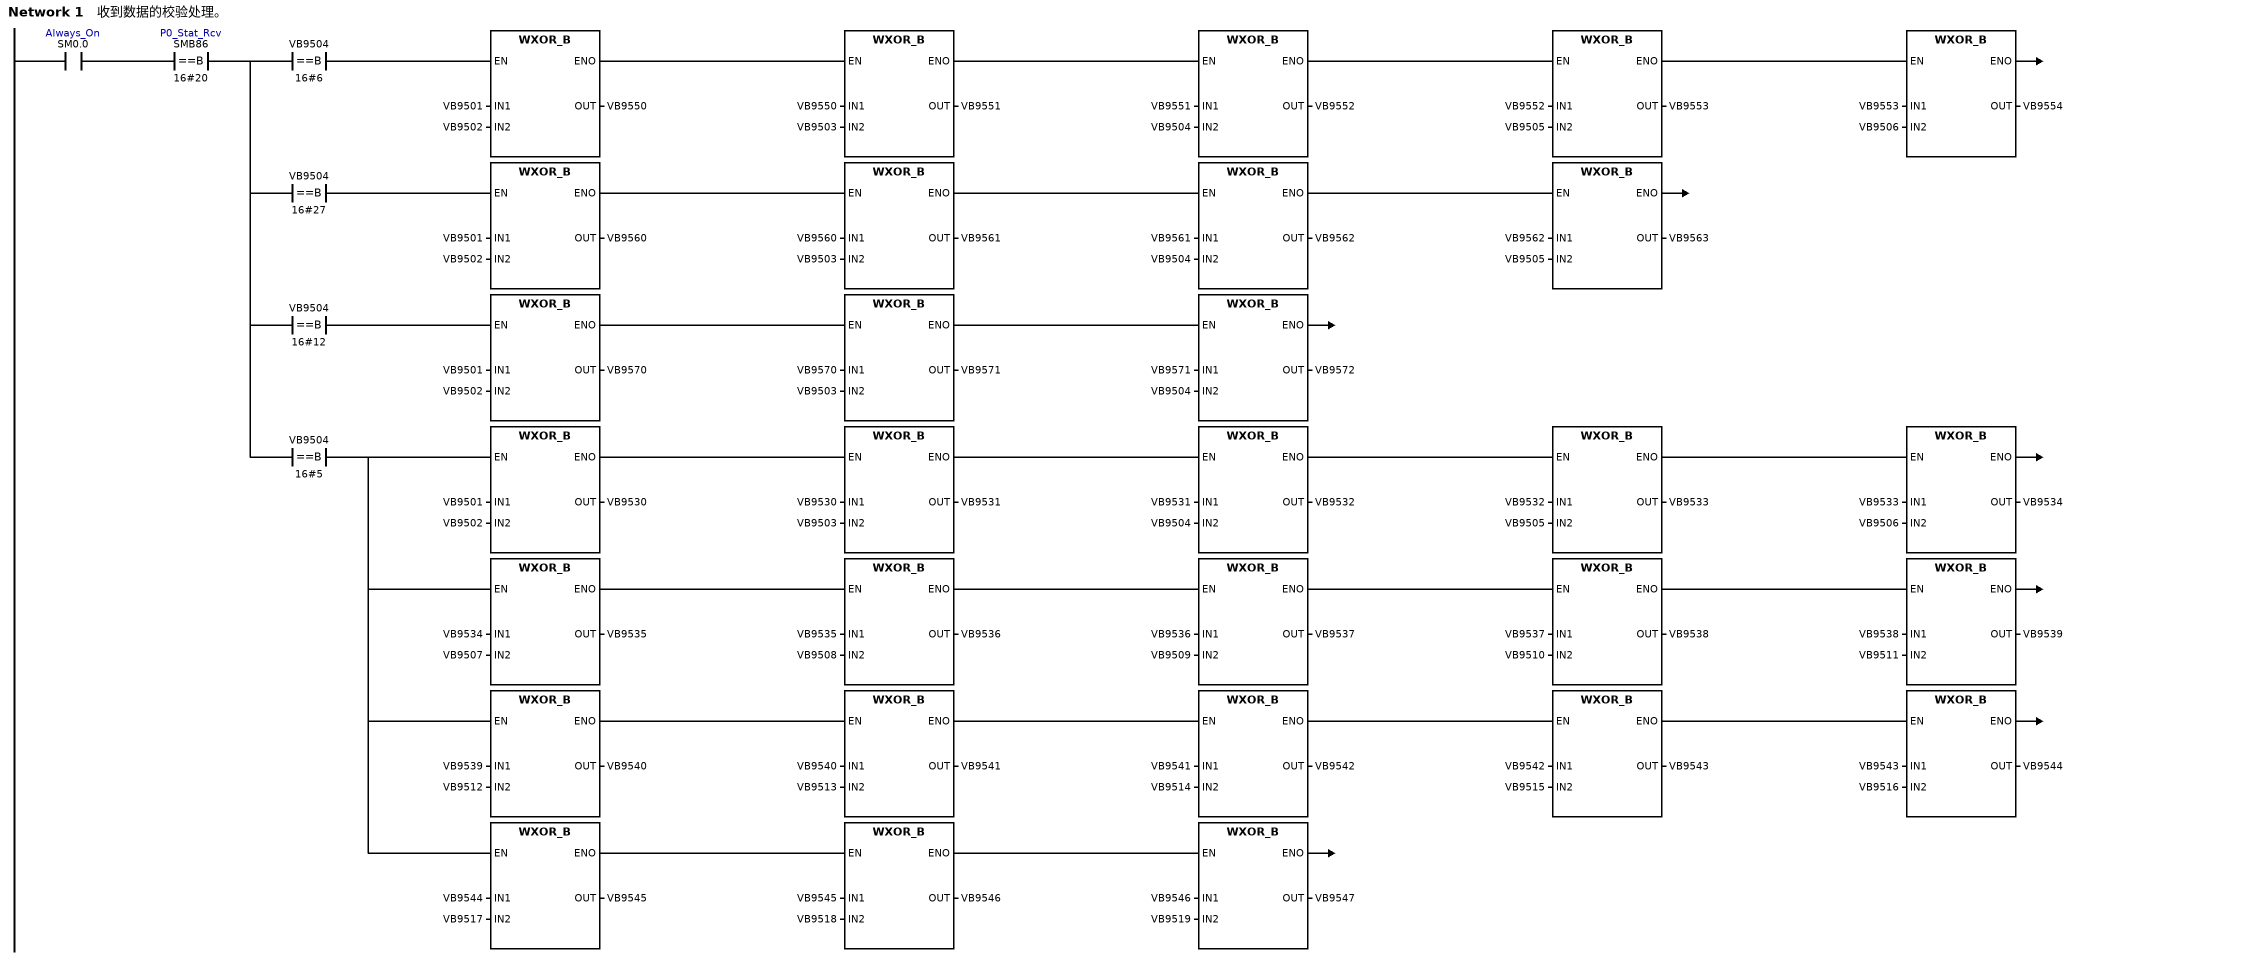
Network 1 //  收到数据的校验处理。
LD     Always_On:SM0.0
AB=    P0_Stat_Rcv:SMB86, 16#20
LPS
AB=    VB9504, 16#6
MOVB   VB9501, VB9550
AENO
XORB   VB9502, VB9550
AENO
MOVB   VB9550, VB9551
AENO
XORB   VB9503, VB9551
AENO
MOVB   VB9551, VB9552
AENO
XORB   VB9504, VB9552
AENO
MOVB   VB9552, VB9553
AENO
XORB   VB9505, VB9553
AENO
MOVB   VB9553, VB9554
XORB   VB9506, VB9554
LRD
AB=    VB9504, 16#27
MOVB   VB9501, VB9560
AENO
XORB   VB9502, VB9560
AENO
MOVB   VB9560, VB9561
AENO
XORB   VB9503, VB9561
AENO
MOVB   VB9561, VB9562
AENO
XORB   VB9504, VB9562
AENO
MOVB   VB9562, VB9563
XORB   VB9505, VB9563
LRD
AB=    VB9504, 16#12
MOVB   VB9501, VB9570
AENO
XORB   VB9502, VB9570
AENO
MOVB   VB9570, VB9571
AENO
XORB   VB9503, VB9571
AENO
MOVB   VB9571, VB9572
XORB   VB9504, VB9572
LPP
AB=    VB9504, 16#5
LPS
MOVB   VB9501, VB9530
AENO
XORB   VB9502, VB9530
AENO
MOVB   VB9530, VB9531
AENO
XORB   VB9503, VB9531
AENO
MOVB   VB9531, VB9532
AENO
XORB   VB9504, VB9532
AENO
MOVB   VB9532, VB9533
AENO
XORB   VB9505, VB9533
AENO
MOVB   VB9533, VB9534
XORB   VB9506, VB9534
LRD
MOVB   VB9534, VB9535
AENO
XORB   VB9507, VB9535
AENO
MOVB   VB9535, VB9536
AENO
XORB   VB9508, VB9536
AENO
MOVB   VB9536, VB9537
AENO
XORB   VB9509, VB9537
AENO
MOVB   VB9537, VB9538
AENO
XORB   VB9510, VB9538
AENO
MOVB   VB9538, VB9539
XORB   VB9511, VB9539
LRD
MOVB   VB9539, VB9540
AENO
XORB   VB9512, VB9540
AENO
MOVB   VB9540, VB9541
AENO
XORB   VB9513, VB9541
AENO
MOVB   VB9541, VB9542
AENO
XORB   VB9514, VB9542
AENO
MOVB   VB9542, VB9543
AENO
XORB   VB9515, VB9543
AENO
MOVB   VB9543, VB9544
XORB   VB9516, VB9544
LPP
MOVB   VB9544, VB9545
AENO
XORB   VB9517, VB9545
AENO
MOVB   VB9545, VB9546
AENO
XORB   VB9518, VB9546
AENO
MOVB   VB9546, VB9547
XORB   VB9519, VB9547
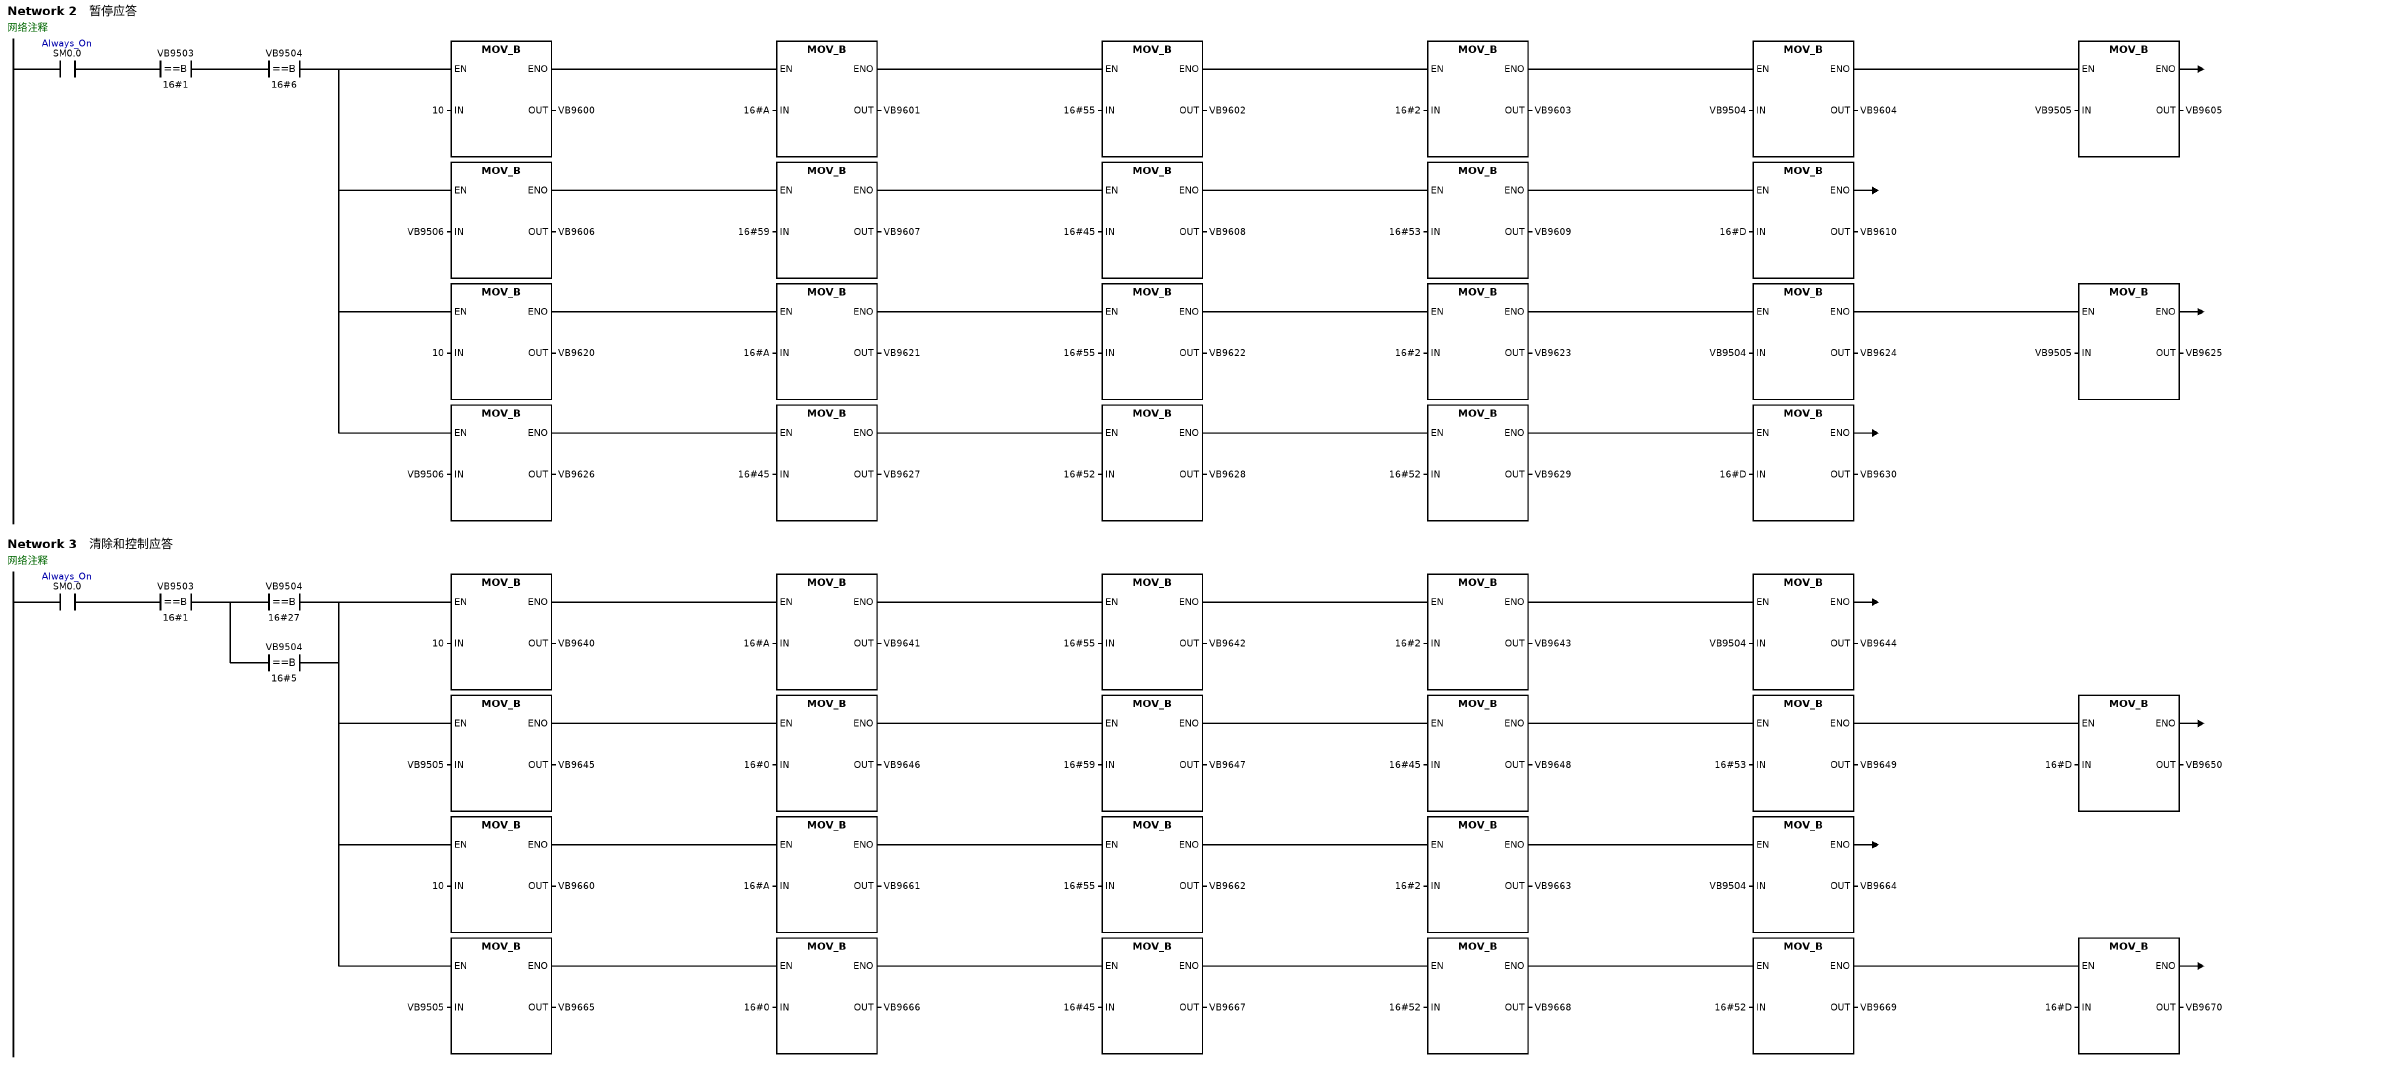
Network 2 //  暂停应答
//  网络注释
LD     Always_On:SM0.0
AB=    VB9503, 16#1
AB=    VB9504, 16#6
LPS
MOVB   10, VB9600
AENO
MOVB   16#A, VB9601
AENO
MOVB   16#55, VB9602
AENO
MOVB   16#2, VB9603
AENO
MOVB   VB9504, VB9604
AENO
MOVB   VB9505, VB9605
LRD
MOVB   VB9506, VB9606
AENO
MOVB   16#59, VB9607
AENO
MOVB   16#45, VB9608
AENO
MOVB   16#53, VB9609
AENO
MOVB   16#D, VB9610
LRD
MOVB   10, VB9620
AENO
MOVB   16#A, VB9621
AENO
MOVB   16#55, VB9622
AENO
MOVB   16#2, VB9623
AENO
MOVB   VB9504, VB9624
AENO
MOVB   VB9505, VB9625
LPP
MOVB   VB9506, VB9626
AENO
MOVB   16#45, VB9627
AENO
MOVB   16#52, VB9628
AENO
MOVB   16#52, VB9629
AENO
MOVB   16#D, VB9630
Network 3 //  清除和控制应答
//  网络注释
LD     Always_On:SM0.0
AB=    VB9503, 16#1
LDB=   VB9504, 16#27
OB=    VB9504, 16#5
ALD
LPS
MOVB   10, VB9640
AENO
MOVB   16#A, VB9641
AENO
MOVB   16#55, VB9642
AENO
MOVB   16#2, VB9643
AENO
MOVB   VB9504, VB9644
LRD
MOVB   VB9505, VB9645
AENO
MOVB   16#0, VB9646
AENO
MOVB   16#59, VB9647
AENO
MOVB   16#45, VB9648
AENO
MOVB   16#53, VB9649
AENO
MOVB   16#D, VB9650
LRD
MOVB   10, VB9660
AENO
MOVB   16#A, VB9661
AENO
MOVB   16#55, VB9662
AENO
MOVB   16#2, VB9663
AENO
MOVB   VB9504, VB9664
LPP
MOVB   VB9505, VB9665
AENO
MOVB   16#0, VB9666
AENO
MOVB   16#45, VB9667
AENO
MOVB   16#52, VB9668
AENO
MOVB   16#52, VB9669
AENO
MOVB   16#D, VB9670
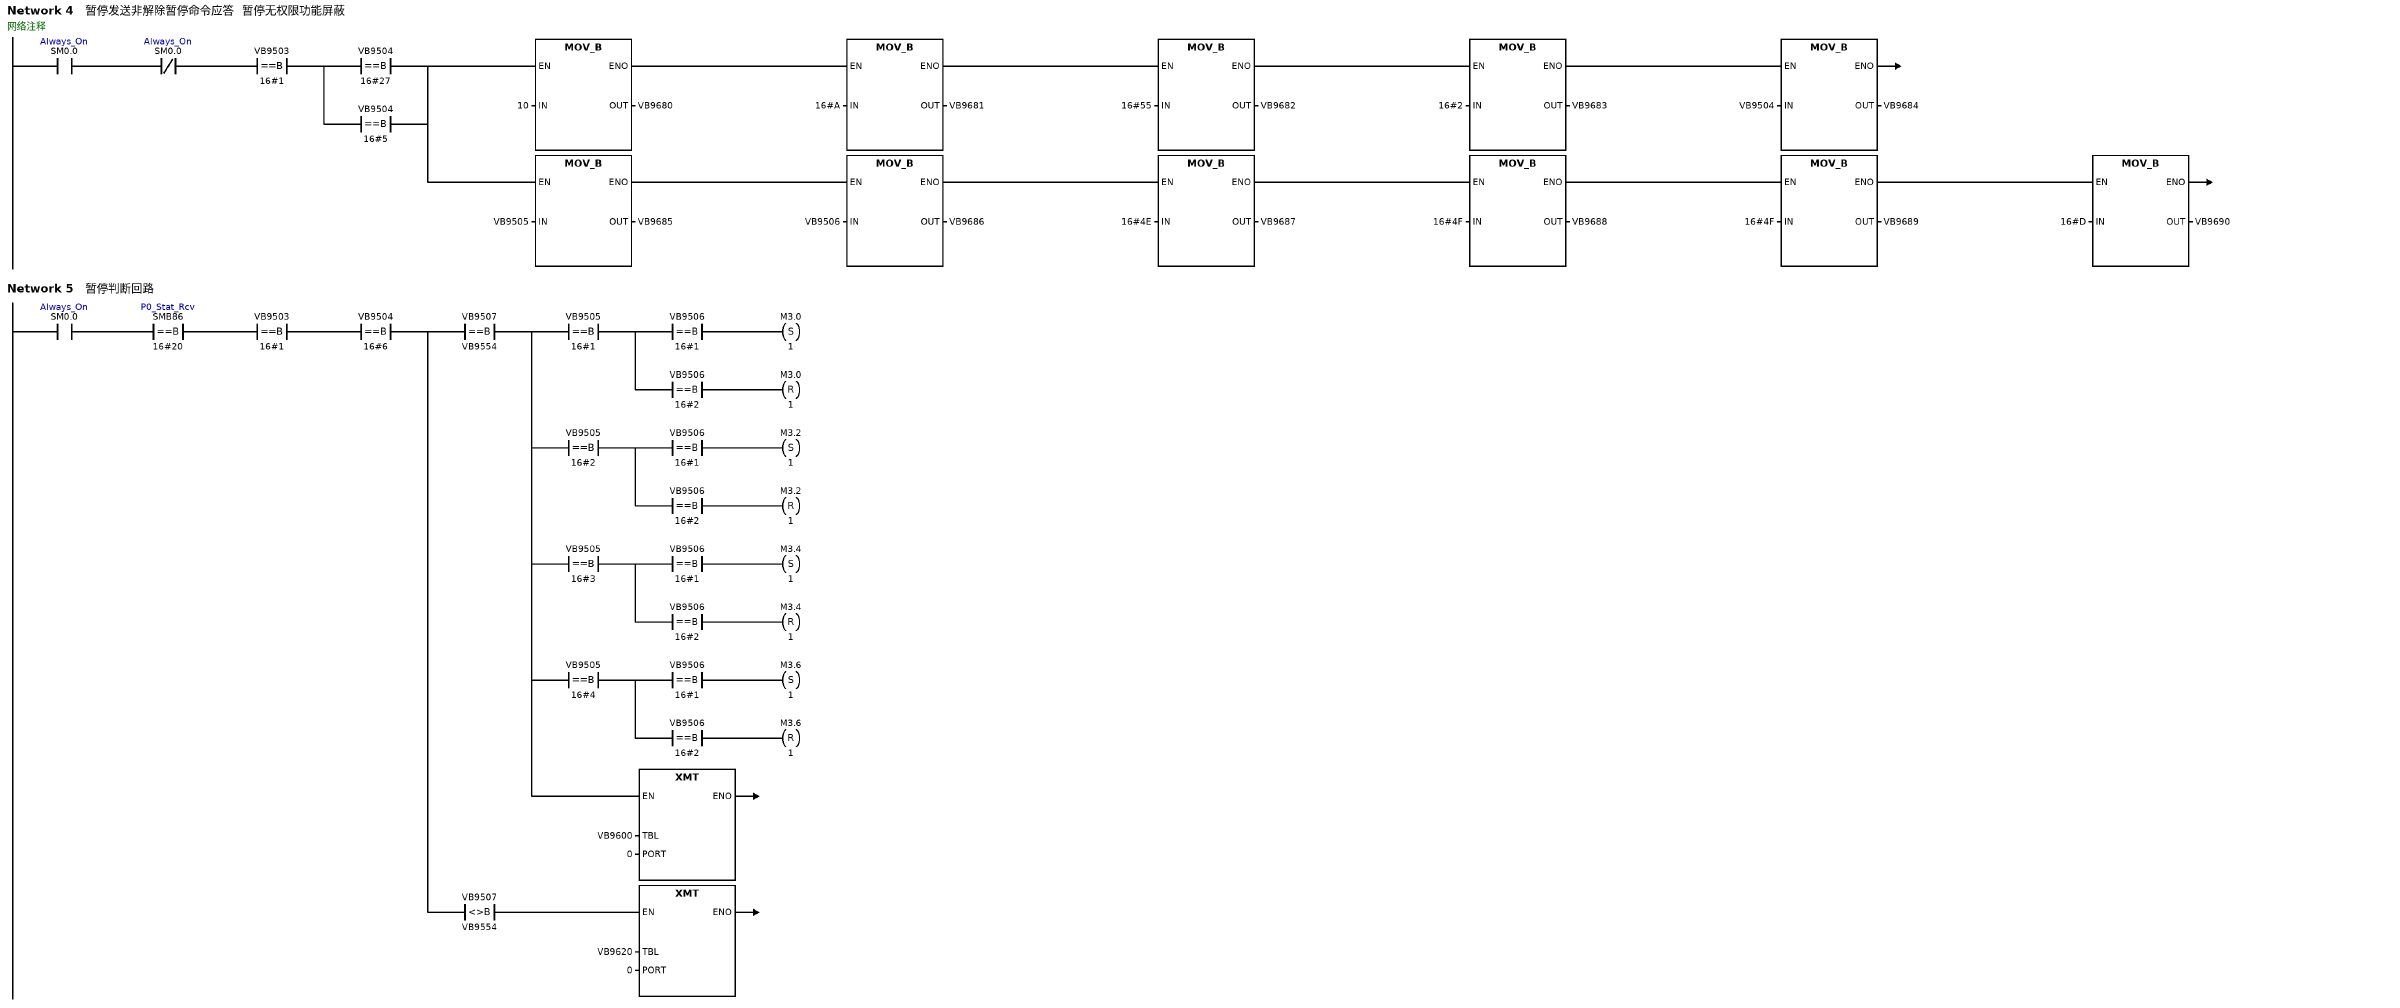
Network 4 //  暂停发送非解除暂停命令应答  暂停无权限功能屏蔽
//  网络注释
LD     Always_On:SM0.0
AN     Always_On:SM0.0
AB=    VB9503, 16#1
LDB=   VB9504, 16#27
OB=    VB9504, 16#5
ALD
LPS
MOVB   10, VB9680
AENO
MOVB   16#A, VB9681
AENO
MOVB   16#55, VB9682
AENO
MOVB   16#2, VB9683
AENO
MOVB   VB9504, VB9684
LPP
MOVB   VB9505, VB9685
AENO
MOVB   VB9506, VB9686
AENO
MOVB   16#4E, VB9687
AENO
MOVB   16#4F, VB9688
AENO
MOVB   16#4F, VB9689
AENO
MOVB   16#D, VB9690
Network 5 //  暂停判断回路
LD     Always_On:SM0.0
AB=    P0_Stat_Rcv:SMB86, 16#20
AB=    VB9503, 16#1
AB=    VB9504, 16#6
LPS
AB=    VB9507, VB9554
LPS
AB=    VB9505, 16#1
LPS
AB=    VB9506, 16#1
S      M3.0, 1
LPP
AB=    VB9506, 16#2
R      M3.0, 1
LRD
AB=    VB9505, 16#2
LPS
AB=    VB9506, 16#1
S      M3.2, 1
LPP
AB=    VB9506, 16#2
R      M3.2, 1
LRD
AB=    VB9505, 16#3
LPS
AB=    VB9506, 16#1
S      M3.4, 1
LPP
AB=    VB9506, 16#2
R      M3.4, 1
LRD
AB=    VB9505, 16#4
LPS
AB=    VB9506, 16#1
S      M3.6, 1
LPP
AB=    VB9506, 16#2
R      M3.6, 1
LPP
XMT    VB9600, 0
LPP
AB<>   VB9507, VB9554
XMT    VB9620, 0
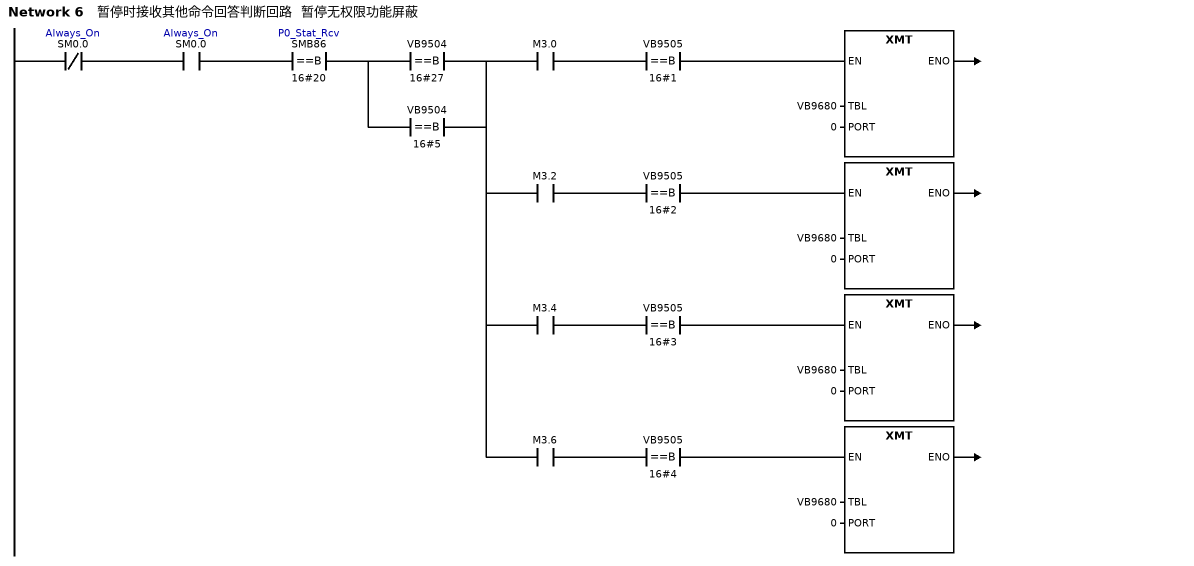
Network 6 //  暂停时接收其他命令回答判断回路  暂停无权限功能屏蔽
LDN    Always_On:SM0.0
A      Always_On:SM0.0
AB=    P0_Stat_Rcv:SMB86, 16#20
LDB=   VB9504, 16#27
OB=    VB9504, 16#5
ALD
LPS
A      M3.0
AB=    VB9505, 16#1
XMT    VB9680, 0
LRD
A      M3.2
AB=    VB9505, 16#2
XMT    VB9680, 0
LRD
A      M3.4
AB=    VB9505, 16#3
XMT    VB9680, 0
LPP
A      M3.6
AB=    VB9505, 16#4
XMT    VB9680, 0
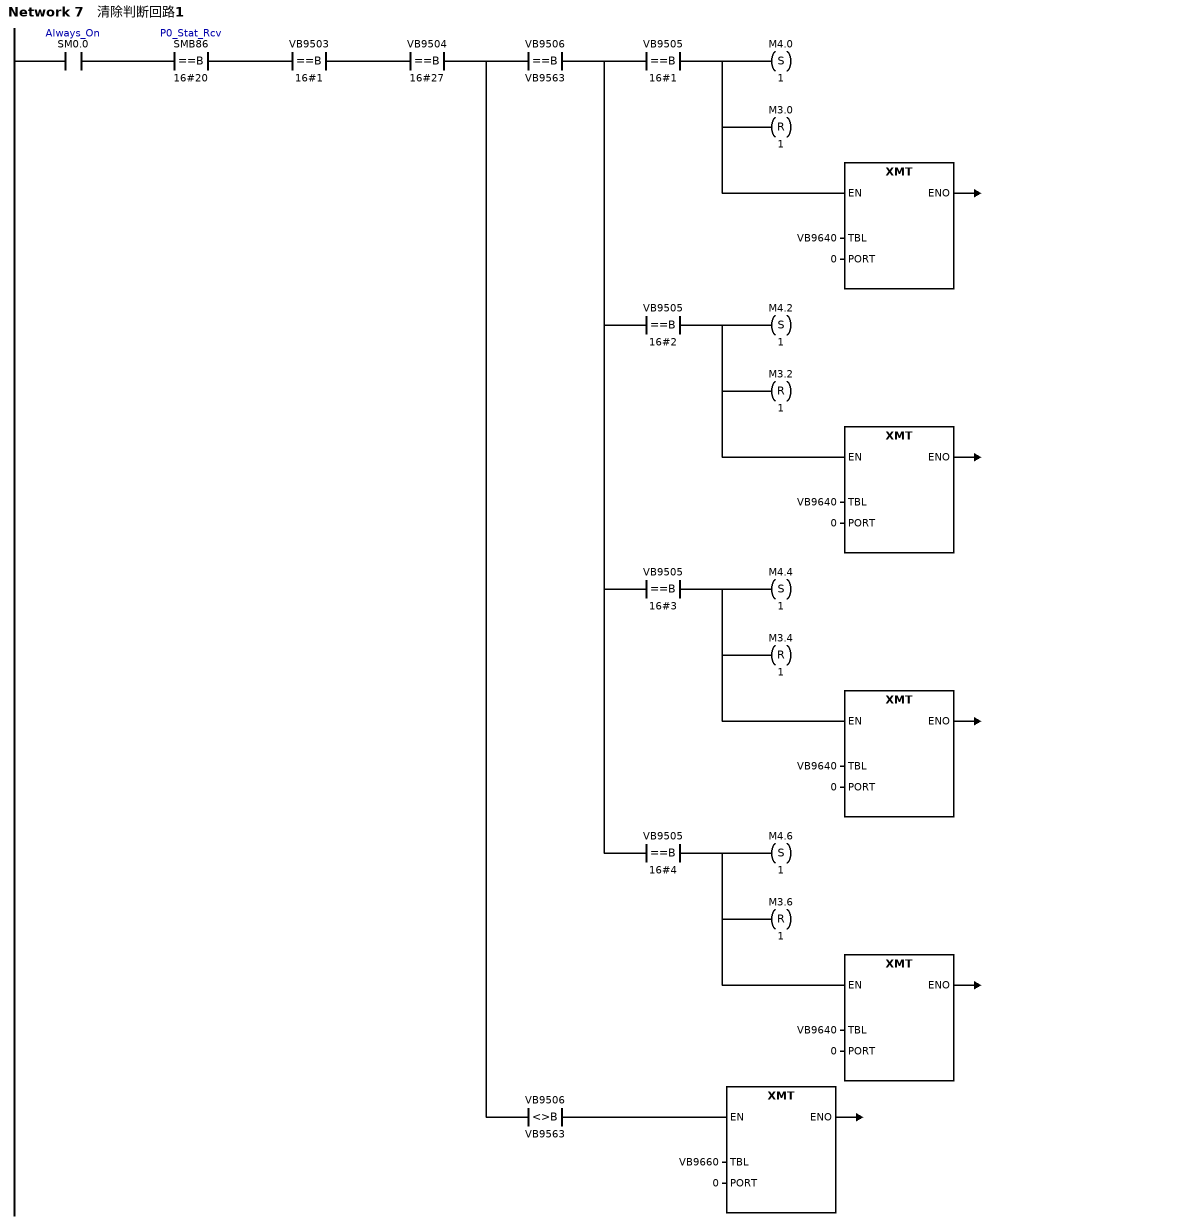
Network 7 //  清除判断回路1
LD     Always_On:SM0.0
AB=    P0_Stat_Rcv:SMB86, 16#20
AB=    VB9503, 16#1
AB=    VB9504, 16#27
LPS
AB=    VB9506, VB9563
LPS
AB=    VB9505, 16#1
S      M4.0, 1
R      M3.0, 1
XMT    VB9640, 0
LRD
AB=    VB9505, 16#2
S      M4.2, 1
R      M3.2, 1
XMT    VB9640, 0
LRD
AB=    VB9505, 16#3
S      M4.4, 1
R      M3.4, 1
XMT    VB9640, 0
LPP
AB=    VB9505, 16#4
S      M4.6, 1
R      M3.6, 1
XMT    VB9640, 0
LPP
AB<>   VB9506, VB9563
XMT    VB9660, 0
Network 8 // 控制判断回路再加一个数据计算判断
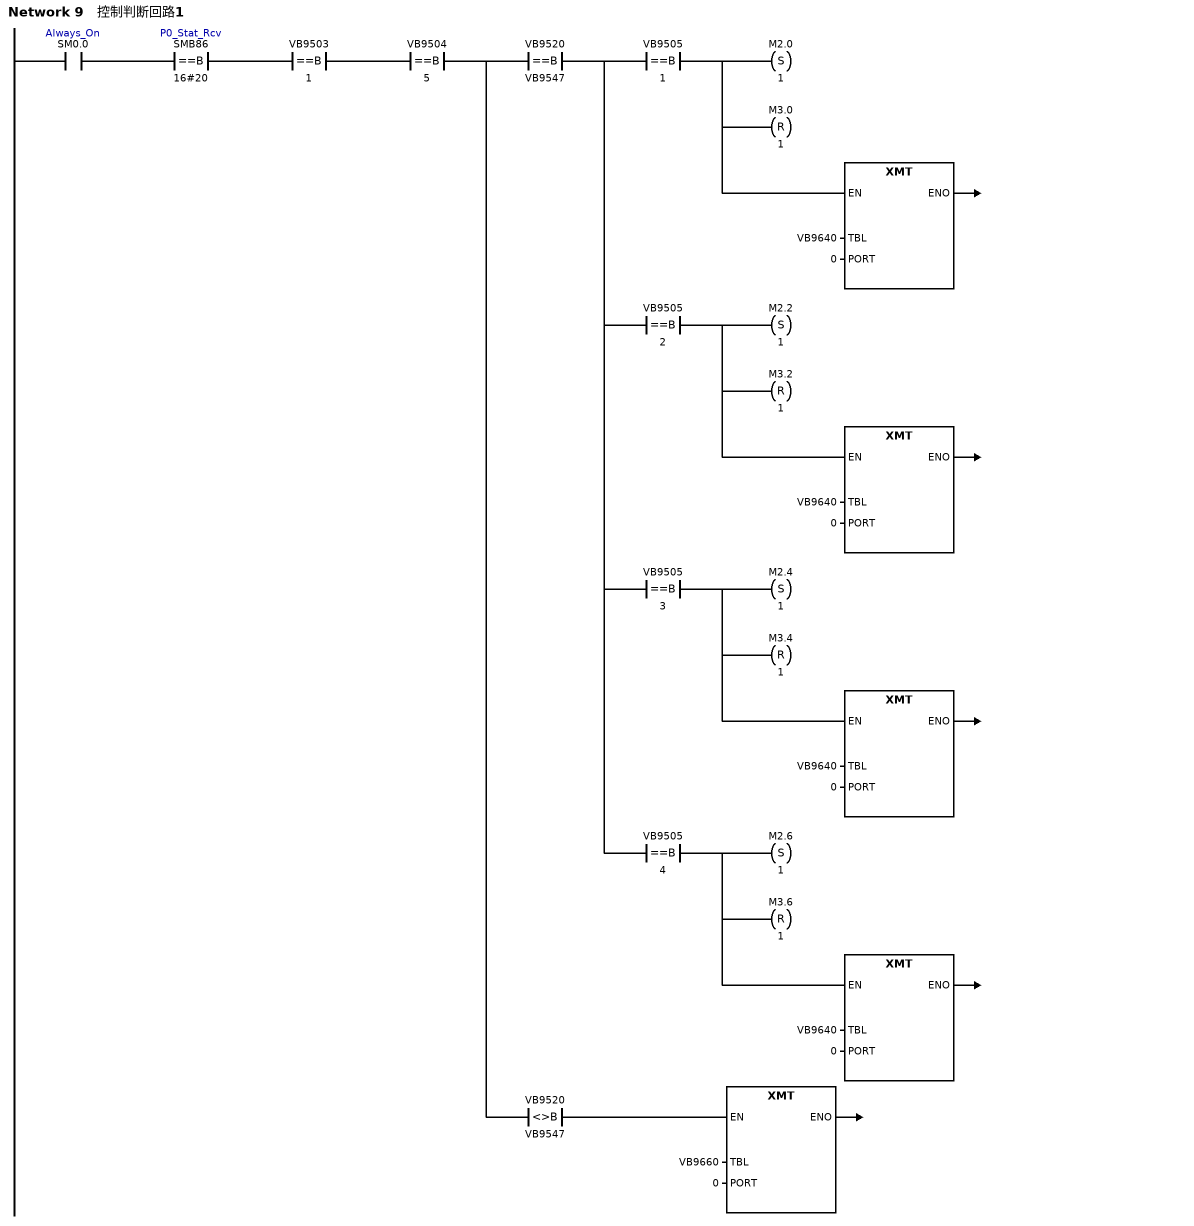
Network 9 //  控制判断回路1
LD     Always_On:SM0.0
AB=    P0_Stat_Rcv:SMB86, 16#20
AB=    VB9503, 1
AB=    VB9504, 5
LPS
AB=    VB9520, VB9547
LPS
AB=    VB9505, 1
S      M2.0, 1
R      M3.0, 1
XMT    VB9640, 0
LRD
AB=    VB9505, 2
S      M2.2, 1
R      M3.2, 1
XMT    VB9640, 0
LRD
AB=    VB9505, 3
S      M2.4, 1
R      M3.4, 1
XMT    VB9640, 0
LPP
AB=    VB9505, 4
S      M2.6, 1
R      M3.6, 1
XMT    VB9640, 0
LPP
AB<>   VB9520, VB9547
XMT    VB9660, 0
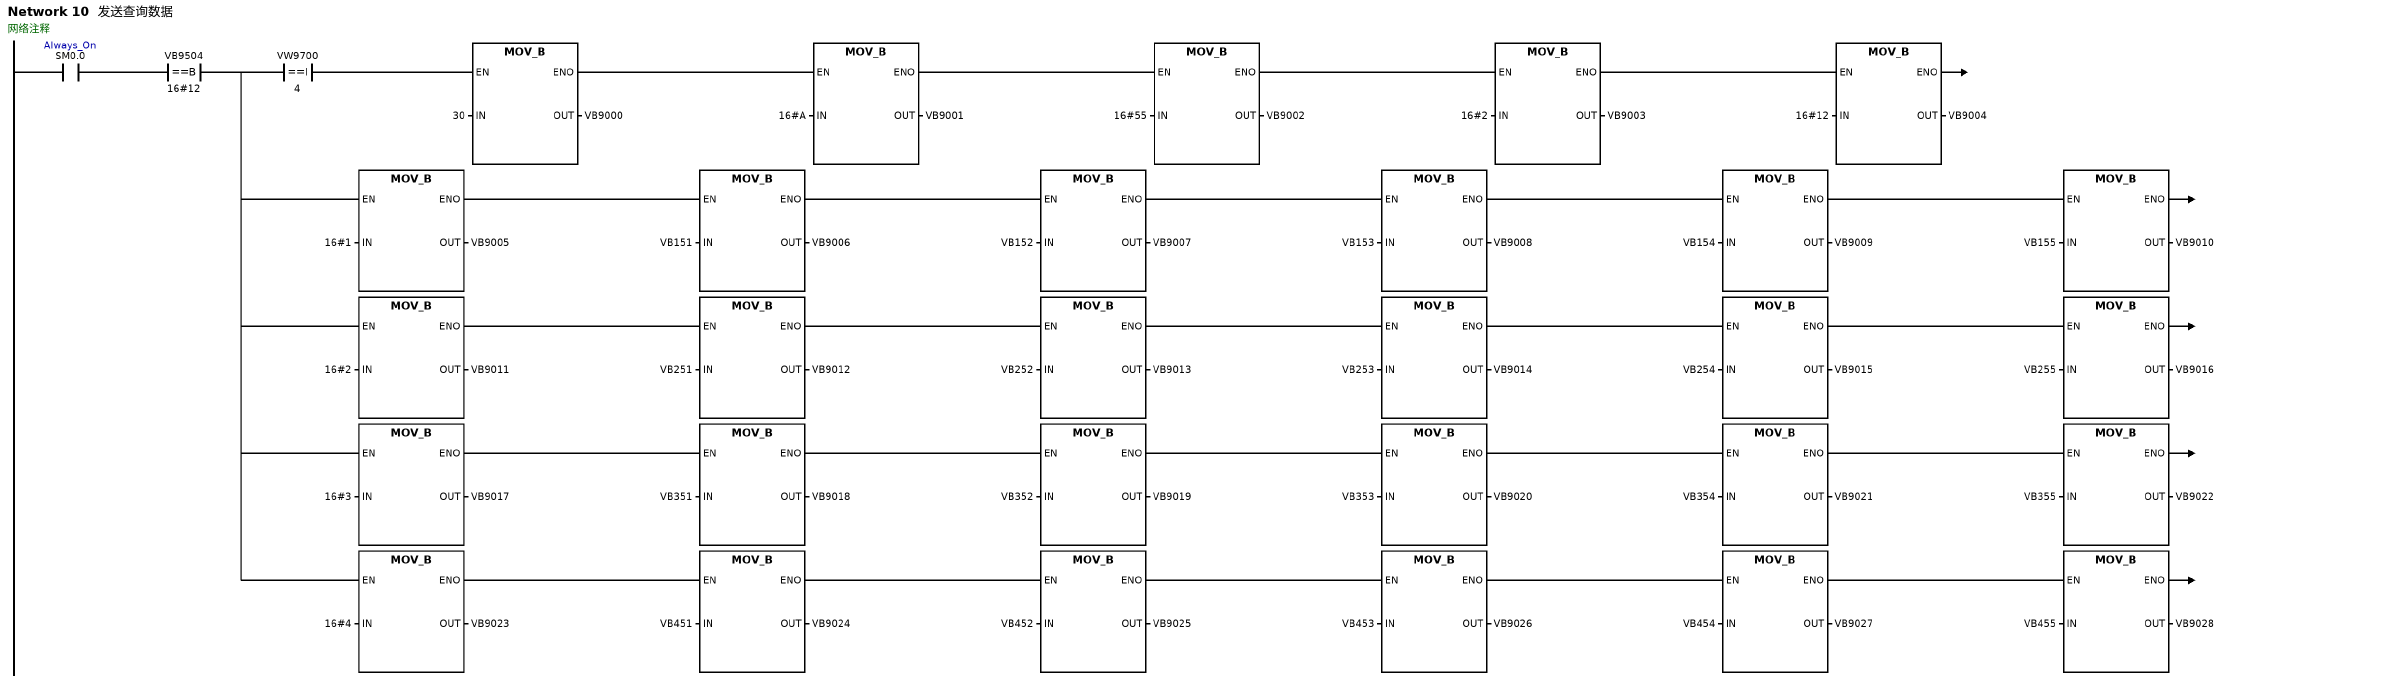
Network 10 // 发送查询数据
// 网络注释
LD     Always_On:SM0.0
AB=    VB9504, 16#12
LPS
AW=    VW9700, 4
MOVB   30, VB9000
AENO
MOVB   16#A, VB9001
AENO
MOVB   16#55, VB9002
AENO
MOVB   16#2, VB9003
AENO
MOVB   16#12, VB9004
LRD
MOVB   16#1, VB9005
AENO
MOVB   VB151, VB9006
AENO
MOVB   VB152, VB9007
AENO
MOVB   VB153, VB9008
AENO
MOVB   VB154, VB9009
AENO
MOVB   VB155, VB9010
LRD
MOVB   16#2, VB9011
AENO
MOVB   VB251, VB9012
AENO
MOVB   VB252, VB9013
AENO
MOVB   VB253, VB9014
AENO
MOVB   VB254, VB9015
AENO
MOVB   VB255, VB9016
LRD
MOVB   16#3, VB9017
AENO
MOVB   VB351, VB9018
AENO
MOVB   VB352, VB9019
AENO
MOVB   VB353, VB9020
AENO
MOVB   VB354, VB9021
AENO
MOVB   VB355, VB9022
LPP
MOVB   16#4, VB9023
AENO
MOVB   VB451, VB9024
AENO
MOVB   VB452, VB9025
AENO
MOVB   VB453, VB9026
AENO
MOVB   VB454, VB9027
AENO
MOVB   VB455, VB9028
